C05498=1143.828,37.027,-50.516,-179.944,6.348,149.136
C05499=1143.823,37.277,-50.531,-179.940,6.350,149.135
C05500=1143.817,37.527,-50.546,-179.938,6.350,149.135
C05501=1143.813,37.776,-50.561,-179.936,6.352,149.135
C05502=1143.807,38.025,-50.576,-179.933,6.353,149.134
C05503=1143.802,38.275,-50.590,-179.930,6.354,149.133
C05504=1143.798,38.524,-50.605,-179.927,6.355,149.133
C05505=1143.792,38.774,-50.620,-179.925,6.355,149.132
C05506=1143.787,39.023,-50.635,-179.923,6.357,149.132
C05507=1143.782,39.272,-50.651,-179.920,6.358,149.131
C05508=1143.777,39.522,-50.665,-179.917,6.359,149.131
C05509=1143.772,39.771,-50.681,-179.915,6.360,149.130
C05510=1143.768,40.021,-50.696,-179.912,6.361,149.130
C05511=1143.762,40.271,-50.711,-179.910,6.362,149.129
C05512=1143.757,40.520,-50.726,-179.906,6.363,149.128
C05513=1143.752,40.770,-50.742,-179.904,6.364,149.128
C05514=1143.747,41.019,-50.757,-179.902,6.365,149.128
C05515=1143.742,41.269,-50.771,-179.899,6.366,149.127
C05516=1143.737,41.518,-50.786,-179.897,6.367,149.126
C05517=1143.732,41.767,-50.802,-179.894,6.369,149.126
C05518=1143.727,42.017,-50.816,-179.891,6.369,149.125
C05519=1143.722,42.267,-50.832,-179.888,6.371,149.125
C05520=1143.717,42.516,-50.847,-179.886,6.371,149.124
C05521=1143.712,42.766,-50.863,-179.883,6.373,149.124
C05522=1143.707,43.015,-50.878,-179.881,6.374,149.123
C05523=1143.701,43.265,-50.893,-179.878,6.375,149.123
C05524=1143.697,43.514,-50.908,-179.876,6.376,149.122
C05525=1143.691,43.763,-50.923,-179.873,6.378,149.122
C05526=1143.687,44.013,-50.939,-179.870,6.378,149.121
C05527=1143.682,44.263,-50.954,-179.868,6.379,149.121
C05528=1143.677,44.512,-50.970,-179.865,6.381,149.120
C05529=1143.672,44.762,-50.984,-179.863,6.381,149.120
C05530=1143.666,45.011,-51.000,-179.860,6.383,149.119
C05531=1143.662,45.260,-51.015,-179.857,6.383,149.118
C05532=1143.657,45.510,-51.031,-179.854,6.385,149.118
C05533=1143.651,45.760,-51.046,-179.852,6.386,149.117
C05534=1143.647,46.009,-51.061,-179.849,6.387,149.117
C05535=1143.641,46.258,-51.077,-179.847,6.388,149.116
C05536=1143.636,46.508,-51.092,-179.844,6.389,149.116
C05537=1143.632,46.757,-51.108,-179.841,6.390,149.115
C05538=1143.627,47.007,-51.123,-179.839,6.391,149.115
C05539=1143.621,47.256,-51.139,-179.837,6.392,149.114
C05540=1143.617,47.505,-51.154,-179.833,6.394,149.114
C05541=1143.611,47.755,-51.169,-179.831,6.394,149.113
C05542=1143.606,48.005,-51.185,-179.828,6.396,149.113
C05543=1143.602,48.254,-51.200,-179.826,6.396,149.112
C05544=1143.596,48.503,-51.216,-179.823,6.398,149.112
C05545=1143.591,48.753,-51.232,-179.820,6.399,149.111
C05546=1143.587,49.002,-51.247,-179.818,6.400,149.111
C05547=1143.582,49.252,-51.263,-179.815,6.401,149.110
C05548=1143.576,49.501,-51.278,-179.812,6.402,149.109
C05549=1143.571,49.750,-51.293,-179.810,6.403,149.109
C05550=1143.567,50.000,-51.309,-179.807,6.405,149.109
C05551=1143.561,50.250,-51.325,-179.805,6.405,149.108
C05552=1143.556,50.499,-51.340,-179.802,6.407,149.107
C05553=1143.551,50.748,-51.355,-179.800,6.408,149.107
C05554=1143.546,50.998,-51.371,-179.796,6.409,149.106
C05555=1143.541,51.248,-51.387,-179.794,6.410,149.106
C05556=1143.536,51.497,-51.402,-179.791,6.411,149.105
C05557=1143.532,51.747,-51.418,-179.789,6.412,149.105
C05558=1143.527,51.996,-51.434,-179.786,6.414,149.104
C05559=1143.521,52.245,-51.450,-179.783,6.415,149.104
C05560=1143.516,52.495,-51.466,-179.781,6.416,149.103
C05561=1143.511,52.745,-51.481,-179.778,6.417,149.103
C05562=1143.506,52.994,-51.496,-179.775,6.418,149.102
C05563=1143.501,53.262,-51.513,-179.773,6.420,149.102
C05564=1143.495,53.531,-51.530,-179.769,6.421,149.101
C05565=1143.490,53.800,-51.548,-179.767,6.422,149.101
C05566=1143.485,54.068,-51.565,-179.764,6.423,149.100
C05567=1143.479,54.318,-51.580,-179.761,6.425,149.099
C05568=1143.475,54.568,-51.596,-179.759,6.425,149.099
C05569=1143.469,54.817,-51.612,-179.756,6.427,149.098
C05570=1143.464,55.066,-51.628,-179.754,6.428,149.098
C05571=1143.460,55.316,-51.643,-179.751,6.429,149.098
C05572=1143.455,55.565,-51.659,-179.748,6.430,149.097
C05573=1143.450,55.814,-51.675,-179.746,6.431,149.096
C05574=1143.445,56.064,-51.691,-179.743,6.432,149.096
C05575=1143.439,56.314,-51.707,-179.740,6.433,149.095
C05576=1143.434,56.562,-51.723,-179.737,6.435,149.095
C05577=1143.430,56.812,-51.739,-179.735,6.436,149.094
C05578=1143.424,57.062,-51.755,-179.732,6.437,149.094
C05579=1143.420,57.311,-51.771,-179.730,6.438,149.093
C05580=1143.414,57.561,-51.787,-179.727,6.440,149.093
C05581=1143.409,57.810,-51.802,-179.724,6.440,149.092
C05582=1143.404,58.060,-51.819,-179.722,6.442,149.092
C05583=1143.400,58.309,-51.834,-179.719,6.443,149.091
C05584=1143.395,58.558,-51.851,-179.716,6.444,149.091
C05585=1143.390,58.808,-51.866,-179.714,6.446,149.090
C05586=1143.385,59.057,-51.882,-179.711,6.446,149.090
C05587=1143.380,59.307,-51.899,-179.708,6.448,149.089
C05588=1143.375,59.556,-51.914,-179.706,6.449,149.089
C05589=1143.370,59.805,-51.931,-179.703,6.450,149.088
C05590=1143.365,60.055,-51.946,-179.700,6.451,149.088
C05591=1143.360,60.304,-51.963,-179.698,6.452,149.087
C05592=1143.355,60.554,-51.979,-179.695,6.454,149.087
C05593=1143.350,60.803,-51.995,-179.693,6.454,149.086
C05594=1143.345,61.053,-52.011,-179.690,6.456,149.086
C05595=1143.339,61.302,-52.028,-179.687,6.458,149.085
C05596=1143.334,61.552,-52.044,-179.684,6.458,149.084
C05597=1143.329,61.801,-52.060,-179.682,6.460,149.084
C05598=1143.325,62.051,-52.076,-179.679,6.461,149.084
C05599=1143.319,62.299,-52.092,-179.676,6.462,149.083
C05600=1143.315,62.550,-52.108,-179.673,6.464,149.083
C05601=1143.310,62.798,-52.125,-179.671,6.465,149.082
C05602=1143.305,63.048,-52.141,-179.668,6.466,149.081
C05603=1143.300,63.297,-52.157,-179.666,6.467,149.081
C05604=1143.295,63.547,-52.174,-179.663,6.468,149.081
C05605=1143.290,63.796,-52.189,-179.660,6.470,149.080
C05606=1143.285,64.046,-52.206,-179.658,6.470,149.079
C05607=1143.280,64.295,-52.221,-179.655,6.472,149.079
C05608=1143.275,64.545,-52.239,-179.653,6.473,149.079
C05609=1143.270,64.794,-52.255,-179.650,6.474,149.078
C05610=1143.265,65.044,-52.271,-179.647,6.476,149.077
C05611=1143.260,65.293,-52.288,-179.645,6.477,149.077
C05612=1143.255,65.542,-52.304,-179.642,6.478,149.076
C05613=1143.251,65.792,-52.320,-179.639,6.480,149.076
C05614=1143.245,66.041,-52.337,-179.637,6.481,149.076
C05615=1143.240,66.291,-52.353,-179.633,6.482,149.075
C05616=1143.235,66.539,-52.370,-179.631,6.483,149.074
C05617=1143.230,66.790,-52.386,-179.629,6.484,149.074
C05618=1143.225,67.038,-52.402,-179.625,6.486,149.073
C05619=1143.221,67.288,-52.419,-179.623,6.486,149.073
C05620=1143.215,67.538,-52.435,-179.620,6.488,149.072
C05621=1143.210,67.787,-52.452,-179.618,6.490,149.072
C05622=1143.206,68.036,-52.468,-179.615,6.490,149.071
C05623=1143.201,68.285,-52.485,-179.612,6.492,149.071
C05624=1143.195,68.535,-52.502,-179.610,6.494,149.070
C05625=1143.191,68.785,-52.518,-179.607,6.494,149.070
C05626=1143.186,69.034,-52.534,-179.604,6.496,149.069
C05627=1143.181,69.283,-52.551,-179.601,6.497,149.069
C05628=1143.175,69.532,-52.568,-179.599,6.498,149.068
C05629=1143.171,69.782,-52.584,-179.596,6.499,149.068
C05630=1143.166,70.031,-52.601,-179.593,6.501,149.067
C05631=1143.161,70.281,-52.617,-179.591,6.502,149.067
C05632=1143.156,70.531,-52.634,-179.588,6.503,149.066
C05633=1143.151,70.780,-52.650,-179.586,6.504,149.066
C05634=1143.146,71.029,-52.667,-179.583,6.506,149.065
C05635=1143.141,71.279,-52.684,-179.580,6.507,149.065
C05636=1143.136,71.528,-52.701,-179.578,6.508,149.064
C05637=1143.131,71.777,-52.717,-179.575,6.510,149.064
C05638=1143.126,72.027,-52.734,-179.572,6.511,149.064
C05639=1143.122,72.276,-52.751,-179.569,6.513,149.063
C05640=1143.117,72.525,-52.767,-179.567,6.513,149.062
C05641=1143.111,72.775,-52.785,-179.564,6.515,149.062
C05642=1143.107,73.024,-52.801,-179.561,6.516,149.061
C05643=1143.102,73.273,-52.817,-179.559,6.517,149.061
C05644=1143.097,73.523,-52.835,-179.556,6.519,149.060
C05645=1143.092,73.772,-52.851,-179.553,6.521,149.060
C05646=1143.086,74.021,-52.868,-179.551,6.521,149.059
C05647=1143.082,74.271,-52.885,-179.548,6.523,149.059
C05648=1143.077,74.520,-52.902,-179.545,6.524,149.059
C05649=1143.072,74.770,-52.919,-179.543,6.525,149.058
C05650=1143.067,75.019,-52.935,-179.540,6.526,149.057
C05651=1143.062,75.269,-52.952,-179.537,6.528,149.057
C05652=1143.057,75.518,-52.969,-179.535,6.529,149.057
C05653=1143.052,75.767,-52.986,-179.532,6.530,149.056
C05654=1143.047,76.017,-53.003,-179.529,6.532,149.056
C05655=1143.043,76.266,-53.019,-179.526,6.534,149.055
C05656=1143.037,76.516,-53.037,-179.524,6.534,149.055
C05657=1143.032,76.765,-53.053,-179.521,6.536,149.054
C05658=1143.027,77.014,-53.071,-179.518,6.537,149.054
C05659=1143.023,77.264,-53.088,-179.516,6.538,149.053
C05660=1143.018,77.513,-53.105,-179.513,6.540,149.053
C05661=1143.013,77.762,-53.121,-179.510,6.541,149.052
C05662=1143.007,78.012,-53.138,-179.508,6.542,149.052
C05663=1143.003,78.261,-53.155,-179.505,6.544,149.051
C05664=1142.998,78.511,-53.173,-179.502,6.545,149.051
C05665=1142.993,78.759,-53.189,-179.499,6.547,149.050
C05666=1142.988,79.009,-53.207,-179.497,6.548,149.050
C05667=1142.982,79.278,-53.225,-179.494,6.549,149.049
C05668=1142.977,79.546,-53.243,-179.491,6.551,149.049
C05669=1142.972,79.815,-53.262,-179.488,6.552,149.048
C05670=1142.967,80.083,-53.281,-179.485,6.554,149.048
C05671=1142.962,80.333,-53.298,-179.482,6.555,149.047
C05672=1142.956,80.582,-53.315,-179.479,6.557,149.047
C05673=1142.952,80.831,-53.331,-179.477,6.558,149.046
C05674=1142.947,81.080,-53.349,-179.474,6.559,149.046
C05675=1142.942,81.330,-53.366,-179.471,6.561,149.045
C05676=1142.937,81.580,-53.383,-179.469,6.562,149.045
C05677=1142.932,81.829,-53.401,-179.466,6.563,149.044
C05678=1142.927,82.078,-53.418,-179.463,6.564,149.044
C05679=1142.922,82.327,-53.435,-179.460,6.566,149.043
C05680=1142.917,82.577,-53.453,-179.458,6.568,149.043
C05681=1142.913,82.826,-53.470,-179.456,6.569,149.042
C05682=1142.907,83.076,-53.487,-179.452,6.570,149.042
C05683=1142.903,83.325,-53.504,-179.450,6.572,149.041
C05684=1142.898,83.574,-53.521,-179.447,6.573,149.041
C05685=1142.892,83.823,-53.539,-179.445,6.574,149.040
C05686=1142.888,84.072,-53.556,-179.441,6.575,149.040
C05687=1142.883,84.322,-53.574,-179.439,6.577,149.039
C05688=1142.878,84.571,-53.591,-179.436,6.579,149.039
C05689=1142.873,84.821,-53.609,-179.434,6.580,149.039
C05690=1142.868,85.070,-53.626,-179.431,6.581,149.038
C05691=1142.863,85.320,-53.643,-179.428,6.583,149.037
C05692=1142.858,85.569,-53.661,-179.425,6.584,149.037
C05693=1142.854,85.819,-53.678,-179.423,6.585,149.037
C05694=1142.849,86.068,-53.696,-179.420,6.586,149.036
C05695=1142.844,86.317,-53.713,-179.417,6.588,149.036
C05696=1142.838,86.566,-53.730,-179.414,6.590,149.035
C05697=1142.834,86.815,-53.748,-179.412,6.591,149.035
C05698=1142.829,87.065,-53.765,-179.409,6.592,149.034
C05699=1142.824,87.314,-53.783,-179.406,6.594,149.034
C05700=1142.819,87.564,-53.800,-179.403,6.595,149.033
C05701=1142.814,87.813,-53.818,-179.401,6.597,149.033
C05702=1142.809,88.062,-53.835,-179.399,6.598,149.032
C05703=1142.804,88.311,-53.853,-179.395,6.599,149.032
C05704=1142.799,88.561,-53.871,-179.393,6.601,149.031
C05705=1142.794,88.810,-53.888,-179.390,6.603,149.031
C05706=1142.789,89.060,-53.906,-179.387,6.604,149.030
C05707=1142.785,89.308,-53.924,-179.385,6.605,149.030
C05708=1142.780,89.558,-53.941,-179.382,6.606,149.029
C05709=1142.775,89.807,-53.959,-179.379,6.608,149.029
C05710=1142.770,90.057,-53.977,-179.376,6.610,149.029
C05711=1142.765,90.306,-53.994,-179.374,6.611,149.028
C05712=1142.760,90.556,-54.012,-179.371,6.612,149.028
C05713=1142.755,90.805,-54.030,-179.368,6.614,149.027
C05714=1142.751,91.054,-54.047,-179.365,6.615,149.027
C05715=1142.746,91.303,-54.065,-179.363,6.617,149.026
C05716=1142.741,91.553,-54.083,-179.360,6.619,149.026
C05717=1142.736,91.802,-54.101,-179.357,6.620,149.025
C05718=1142.731,92.052,-54.118,-179.355,6.621,149.025
C05719=1142.726,92.301,-54.136,-179.352,6.622,149.024
C05720=1142.721,92.550,-54.154,-179.349,6.624,149.024
C05721=1142.716,92.799,-54.172,-179.346,6.626,149.023
C05722=1142.711,93.048,-54.190,-179.344,6.627,149.023
C05723=1142.706,93.298,-54.207,-179.341,6.628,149.022
C05724=1142.701,93.548,-54.225,-179.338,6.630,149.022
C05725=1142.697,93.797,-54.243,-179.336,6.631,149.022
C05726=1142.692,94.046,-54.261,-179.333,6.633,149.021
C05727=1142.687,94.295,-54.279,-179.330,6.635,149.021
C05728=1142.683,94.544,-54.297,-179.327,6.636,149.020
C05729=1142.678,94.793,-54.315,-179.324,6.638,149.020
C05730=1142.672,95.043,-54.332,-179.322,6.638,149.019
C05731=1142.668,95.292,-54.350,-179.319,6.640,149.019
C05732=1142.663,95.542,-54.368,-179.317,6.642,149.018
C05733=1142.657,95.791,-54.386,-179.313,6.643,149.018
C05734=1142.652,96.040,-54.404,-179.311,6.645,149.017
C05735=1142.648,96.290,-54.423,-179.308,6.646,149.017
C05736=1142.643,96.539,-54.441,-179.306,6.647,149.016
C05737=1142.638,96.789,-54.459,-179.303,6.649,149.016
C05738=1142.633,97.038,-54.477,-179.300,6.651,149.016
C05739=1142.628,97.287,-54.495,-179.297,6.652,149.015
C05740=1142.623,97.536,-54.513,-179.294,6.654,149.015
C05741=1142.618,97.785,-54.531,-179.292,6.655,149.014
C05742=1142.614,98.035,-54.549,-179.289,6.657,149.014
C05743=1142.609,98.284,-54.567,-179.287,6.658,149.013
C05744=1142.604,98.533,-54.585,-179.283,6.659,149.013
C05745=1142.599,98.783,-54.603,-179.281,6.661,149.012
C05746=1142.594,99.032,-54.621,-179.278,6.663,149.012
C05747=1142.589,99.281,-54.640,-179.275,6.664,149.011
C05748=1142.584,99.531,-54.658,-179.273,6.666,149.011
C05749=1142.579,99.780,-54.676,-179.270,6.668,149.011
C05750=1142.575,100.030,-54.694,-179.267,6.669,149.010
C05751=1142.570,100.278,-54.713,-179.264,6.670,149.010
C05752=1142.565,100.527,-54.730,-179.262,6.671,149.009
C05753=1142.560,100.776,-54.748,-179.259,6.673,149.009
C05754=1142.555,101.027,-54.767,-179.256,6.675,149.008
C05755=1142.550,101.276,-54.785,-179.253,6.677,149.008
C05756=1142.545,101.525,-54.803,-179.251,6.678,149.007
C05757=1142.540,101.774,-54.821,-179.248,6.680,149.007
C05758=1142.536,102.023,-54.840,-179.245,6.681,149.006
C05759=1142.531,102.273,-54.859,-179.242,6.683,149.006
C05760=1142.526,102.522,-54.877,-179.240,6.684,149.006
C05761=1142.521,102.771,-54.895,-179.237,6.685,149.005
C05762=1142.517,103.020,-54.914,-179.234,6.687,149.005
C05763=1142.512,103.270,-54.932,-179.231,6.688,149.004
C05764=1142.506,103.519,-54.951,-179.229,6.690,149.004
C05765=1142.501,103.768,-54.969,-179.226,6.692,149.003
C05766=1142.497,104.018,-54.988,-179.223,6.693,149.003
C05767=1142.492,104.267,-55.006,-179.220,6.695,149.002
C05768=1142.487,104.516,-55.024,-179.218,6.697,149.002
C05769=1142.482,104.765,-55.042,-179.215,6.699,149.002
C05770=1142.478,105.015,-55.061,-179.212,6.700,149.001
C05771=1142.472,105.283,-55.081,-179.209,6.702,149.001
C05772=1142.467,105.551,-55.101,-179.206,6.703,149.000
C05773=1142.461,105.819,-55.121,-179.203,6.705,149.000
C05774=1142.456,106.088,-55.141,-179.200,6.706,148.999
C05775=1142.451,106.338,-55.160,-179.198,6.708,148.999
C05776=1142.447,106.586,-55.178,-179.195,6.710,148.998
C05777=1142.442,106.836,-55.196,-179.192,6.711,148.998
C05778=1142.437,107.086,-55.215,-179.189,6.713,148.998
C05779=1142.432,107.334,-55.234,-179.187,6.715,148.997
C05780=1142.427,107.584,-55.252,-179.183,6.716,148.996
C05781=1142.422,107.833,-55.272,-179.181,6.718,148.996
C05782=1142.418,108.082,-55.290,-179.178,6.719,148.996
C05783=1142.413,108.331,-55.308,-179.175,6.721,148.995
C05784=1142.408,108.581,-55.327,-179.172,6.723,148.995
C05785=1142.403,108.830,-55.346,-179.170,6.724,148.994
C05786=1142.398,109.080,-55.365,-179.168,6.725,148.994
C05787=1142.394,109.328,-55.384,-179.165,6.727,148.994
C05788=1142.388,109.578,-55.402,-179.162,6.729,148.993
C05789=1142.384,109.827,-55.421,-179.159,6.730,148.993
C05790=1142.379,110.076,-55.439,-179.156,6.732,148.992
C05791=1142.374,110.325,-55.458,-179.153,6.733,148.992
C05792=1142.369,110.575,-55.477,-179.151,6.735,148.991
C05793=1142.364,110.824,-55.496,-179.148,6.737,148.991
C05794=1142.360,111.074,-55.514,-179.145,6.738,148.991
C05795=1142.354,111.323,-55.534,-179.143,6.740,148.990
C05796=1142.350,111.571,-55.552,-179.140,6.742,148.990
C05797=1142.345,111.821,-55.571,-179.137,6.743,148.989
C05798=1142.340,112.070,-55.590,-179.134,6.745,148.989
C05799=1142.335,112.319,-55.610,-179.131,6.746,148.988
C05800=1142.331,112.569,-55.628,-179.128,6.748,148.988
C05801=1142.326,112.818,-55.647,-179.126,6.750,148.987
C05802=1142.321,113.067,-55.665,-179.123,6.751,148.987
C05803=1142.316,113.316,-55.685,-179.120,6.753,148.987
C05804=1142.312,113.565,-55.704,-179.118,6.755,148.986
C05805=1142.306,113.814,-55.723,-179.115,6.757,148.986
C05806=1142.301,114.065,-55.742,-179.112,6.758,148.985
C05807=1142.297,114.313,-55.761,-179.109,6.760,148.985
C05808=1142.292,114.563,-55.780,-179.107,6.762,148.985
C05809=1142.287,114.812,-55.798,-179.103,6.763,148.984
C05810=1142.282,115.061,-55.818,-179.101,6.765,148.984
C05811=1142.277,115.310,-55.837,-179.098,6.766,148.983
C05812=1142.273,115.560,-55.856,-179.095,6.768,148.983
C05813=1142.267,115.808,-55.876,-179.093,6.770,148.982
C05814=1142.263,116.058,-55.894,-179.090,6.771,148.982
C05815=1142.258,116.307,-55.913,-179.087,6.773,148.982
C05816=1142.253,116.557,-55.933,-179.084,6.775,148.981
C05817=1142.248,116.805,-55.952,-179.082,6.776,148.981
C05818=1142.244,117.055,-55.971,-179.079,6.778,148.980
C05819=1142.238,117.304,-55.991,-179.076,6.780,148.980
C05820=1142.234,117.554,-56.009,-179.073,6.782,148.979
C05821=1142.229,117.802,-56.028,-179.071,6.783,148.979
C05822=1142.224,118.052,-56.048,-179.068,6.785,148.979
C05823=1142.219,118.301,-56.066,-179.065,6.786,148.978
C05824=1142.215,118.550,-56.086,-179.062,6.788,148.978
C05825=1142.209,118.799,-56.105,-179.059,6.790,148.977
C05826=1142.205,119.048,-56.125,-179.057,6.791,148.977
C05827=1142.201,119.298,-56.144,-179.054,6.793,148.976
C05828=1142.195,119.547,-56.163,-179.051,6.795,148.976
C05829=1142.190,119.796,-56.183,-179.048,6.796,148.976
C05830=1142.186,120.045,-56.202,-179.046,6.798,148.975
C05831=1142.181,120.294,-56.221,-179.043,6.800,148.975
C05832=1142.176,120.543,-56.241,-179.040,6.801,148.974
C05833=1142.171,120.793,-56.260,-179.038,6.803,148.974
C05834=1142.167,121.042,-56.279,-179.035,6.805,148.974
C05835=1142.162,121.291,-56.299,-179.032,6.807,148.973
C05836=1142.157,121.541,-56.318,-179.029,6.808,148.973
C05837=1142.152,121.790,-56.338,-179.027,6.810,148.972
C05838=1142.147,122.039,-56.357,-179.024,6.812,148.972
C05839=1142.143,122.288,-56.376,-179.021,6.813,148.972
C05840=1142.137,122.537,-56.396,-179.018,6.815,148.971
C05841=1142.133,122.787,-56.415,-179.015,6.818,148.971
C05842=1142.128,123.036,-56.435,-179.012,6.819,148.970
C05843=1142.123,123.284,-56.455,-179.010,6.821,148.970
C05844=1142.118,123.534,-56.475,-179.006,6.822,148.969
C05845=1142.114,123.783,-56.494,-179.004,6.824,148.969
C05846=1142.109,124.032,-56.513,-179.001,6.826,148.969
C05847=1142.104,124.282,-56.533,-178.998,6.827,148.968
C05848=1142.099,124.531,-56.552,-178.996,6.829,148.968
C05849=1142.094,124.780,-56.572,-178.993,6.831,148.967
C05850=1142.090,125.029,-56.592,-178.990,6.832,148.967
C05851=1142.085,125.279,-56.612,-178.987,6.834,148.967
C05852=1142.079,125.528,-56.631,-178.985,6.836,148.966
C05853=1142.075,125.777,-56.651,-178.982,6.837,148.966
C05854=1142.071,126.026,-56.670,-178.979,6.839,148.965
C05855=1142.066,126.275,-56.690,-178.976,6.842,148.965
C05856=1142.061,126.524,-56.709,-178.973,6.843,148.965
C05857=1142.057,126.773,-56.730,-178.970,6.845,148.964
C05858=1142.052,127.023,-56.749,-178.968,6.847,148.964
C05859=1142.046,127.272,-56.769,-178.965,6.848,148.963
C05860=1142.042,127.521,-56.788,-178.962,6.850,148.963
C05861=1142.037,127.770,-56.809,-178.960,6.852,148.963
C05862=1142.033,128.020,-56.828,-178.957,6.854,148.962
C05863=1142.027,128.269,-56.848,-178.954,6.855,148.962
C05864=1142.023,128.517,-56.868,-178.951,6.857,148.961
C05865=1142.018,128.767,-56.888,-178.949,6.859,148.961
C05866=1142.014,129.016,-56.908,-178.945,6.861,148.961
C05867=1142.008,129.265,-56.927,-178.943,6.863,148.960
C05868=1142.003,129.514,-56.947,-178.940,6.865,148.960
C05869=1141.999,129.763,-56.967,-178.937,6.866,148.959
C05870=1141.994,130.013,-56.987,-178.935,6.868,148.959
C05871=1141.989,130.261,-57.007,-178.932,6.870,148.959
C05872=1141.985,130.511,-57.027,-178.929,6.871,148.958
C05873=1141.979,130.760,-57.048,-178.926,6.873,148.958
C05874=1141.975,131.010,-57.067,-178.924,6.875,148.957
C05875=1141.970,131.278,-57.088,-178.920,6.877,148.957
C05876=1141.965,131.546,-57.110,-178.918,6.879,148.957
C05877=1141.959,131.815,-57.132,-178.914,6.881,148.956
C05878=1141.954,132.084,-57.153,-178.912,6.883,148.956
C05879=1141.949,132.332,-57.173,-178.909,6.885,148.956
C05880=1141.944,132.582,-57.193,-178.906,6.887,148.955
C05881=1141.940,132.831,-57.214,-178.903,6.888,148.955
C05882=1141.935,133.080,-57.234,-178.901,6.890,148.954
C05883=1141.930,133.329,-57.254,-178.897,6.892,148.954
C05884=1141.926,133.578,-57.274,-178.895,6.894,148.954
C05885=1141.921,133.828,-57.294,-178.892,6.896,148.953
C05886=1141.915,134.077,-57.314,-178.889,6.898,148.953
C05887=1141.911,134.326,-57.335,-178.887,6.899,148.952
C05888=1141.906,134.575,-57.354,-178.884,6.901,148.952
C05889=1141.902,134.824,-57.375,-178.881,6.903,148.952
C05890=1141.897,135.073,-57.395,-178.878,6.905,148.951
C05891=1141.892,135.323,-57.415,-178.875,6.907,148.951
C05892=1141.887,135.572,-57.436,-178.872,6.909,148.950
C05893=1141.883,135.821,-57.456,-178.870,6.910,148.950
C05894=1141.878,136.070,-57.475,-178.867,6.912,148.950
C05895=1141.873,136.319,-57.496,-178.864,6.914,148.949
C05896=1141.868,136.568,-57.517,-178.861,6.915,148.949
C05897=1141.864,136.817,-57.537,-178.859,6.918,148.949
C05898=1141.859,137.066,-57.557,-178.856,6.920,148.948
C05899=1141.854,137.316,-57.578,-178.853,6.922,148.948
C05900=1141.849,137.565,-57.598,-178.850,6.923,148.948
C05901=1141.845,137.814,-57.618,-178.848,6.925,148.947
C05902=1141.840,138.063,-57.638,-178.845,6.927,148.947
C05903=1141.835,138.312,-57.659,-178.842,6.929,148.946
C05904=1141.830,138.561,-57.679,-178.839,6.931,148.946
C05905=1141.826,138.810,-57.700,-178.836,6.933,148.946
C05906=1141.821,139.059,-57.721,-178.834,6.934,148.945
C05907=1141.816,139.308,-57.741,-178.831,6.936,148.945
C05908=1141.812,139.557,-57.761,-178.828,6.939,148.944
C05909=1141.806,139.807,-57.782,-178.825,6.940,148.944
C05910=1141.802,140.056,-57.802,-178.822,6.942,148.944
C05911=1141.797,140.304,-57.822,-178.819,6.944,148.943
C05912=1141.792,140.554,-57.843,-178.817,6.946,148.943
C05913=1141.787,140.803,-57.863,-178.814,6.948,148.943
C05914=1141.782,141.052,-57.884,-178.811,6.950,148.942
C05915=1141.778,141.301,-57.905,-178.808,6.952,148.942
C05916=1141.774,141.551,-57.925,-178.806,6.953,148.942
C05917=1141.769,141.800,-57.946,-178.803,6.955,148.941
C05918=1141.764,142.049,-57.967,-178.800,6.958,148.941
C05919=1141.759,142.298,-57.988,-178.797,6.959,148.940
C05920=1141.755,142.547,-58.008,-178.794,6.961,148.940
C05921=1141.750,142.796,-58.029,-178.792,6.963,148.940
C05922=1141.745,143.045,-58.050,-178.789,6.964,148.939
C05923=1141.741,143.294,-58.070,-178.786,6.967,148.939
C05924=1141.736,143.543,-58.091,-178.783,6.969,148.939
C05925=1141.731,143.792,-58.111,-178.781,6.971,148.938
C05926=1141.726,144.042,-58.132,-178.778,6.972,148.938
C05927=1141.721,144.291,-58.153,-178.775,6.974,148.938
C05928=1141.716,144.540,-58.174,-178.772,6.977,148.937
C05929=1141.712,144.788,-58.195,-178.769,6.978,148.937
C05930=1141.707,145.037,-58.216,-178.766,6.980,148.936
C05931=1141.703,145.286,-58.236,-178.764,6.982,148.936
C05932=1141.697,145.536,-58.257,-178.761,6.985,148.936
C05933=1141.694,145.785,-58.278,-178.758,6.986,148.935
C05934=1141.688,146.034,-58.299,-178.755,6.988,148.935
C05935=1141.683,146.284,-58.320,-178.753,6.990,148.935
C05936=1141.679,146.532,-58.341,-178.749,6.992,148.934
C05937=1141.674,146.781,-58.362,-178.747,6.994,148.934
C05938=1141.669,147.030,-58.382,-178.744,6.996,148.934
C05939=1141.664,147.280,-58.403,-178.741,6.997,148.933
C05940=1141.659,147.528,-58.425,-178.738,7.000,148.933
C05941=1141.655,147.777,-58.445,-178.736,7.002,148.933
C05942=1141.650,148.027,-58.466,-178.733,7.004,148.932
C05943=1141.646,148.276,-58.487,-178.730,7.005,148.932
C05944=1141.641,148.525,-58.508,-178.727,7.008,148.931
C05945=1141.636,148.774,-58.529,-178.724,7.010,148.931
C05946=1141.631,149.023,-58.550,-178.722,7.011,148.931
C05947=1141.627,149.272,-58.571,-178.719,7.014,148.931
C05948=1141.622,149.521,-58.593,-178.716,7.016,148.930
C05949=1141.618,149.770,-58.613,-178.713,7.018,148.930
C05950=1141.613,150.019,-58.635,-178.711,7.019,148.929
C05951=1141.608,150.268,-58.656,-178.708,7.021,148.929
C05952=1141.603,150.517,-58.676,-178.705,7.024,148.929
C05953=1141.598,150.766,-58.698,-178.702,7.025,148.928
C05954=1141.594,151.016,-58.719,-178.700,7.027,148.928
C05955=1141.589,151.265,-58.741,-178.697,7.029,148.928
C05956=1141.584,151.513,-58.761,-178.694,7.032,148.927
C05957=1141.579,151.763,-58.782,-178.691,7.033,148.927
C05958=1141.574,152.011,-58.804,-178.688,7.035,148.927
C05959=1141.570,152.261,-58.825,-178.685,7.038,148.926
C05960=1141.566,152.510,-58.846,-178.683,7.040,148.926
C05961=1141.560,152.759,-58.867,-178.680,7.041,148.926
C05962=1141.556,153.008,-58.889,-178.677,7.043,148.925
C05963=1141.551,153.258,-58.910,-178.674,7.046,148.925
C05964=1141.547,153.506,-58.931,-178.671,7.047,148.925
C05965=1141.542,153.755,-58.952,-178.669,7.049,148.924
C05966=1141.537,154.004,-58.974,-178.666,7.052,148.924
C05967=1141.533,154.253,-58.996,-178.663,7.054,148.924
C05968=1141.527,154.502,-59.017,-178.660,7.055,148.923
C05969=1141.523,154.751,-59.038,-178.657,7.058,148.923
C05970=1141.519,155.001,-59.059,-178.654,7.060,148.923
C05971=1141.514,155.249,-59.081,-178.652,7.062,148.922
C05972=1141.509,155.498,-59.103,-178.649,7.063,148.922
C05973=1141.504,155.747,-59.124,-178.646,7.066,148.922
C05974=1141.499,155.997,-59.146,-178.643,7.068,148.921
C05975=1141.494,156.246,-59.167,-178.641,7.069,148.921
C05976=1141.489,156.494,-59.188,-178.638,7.072,148.921
C05977=1141.486,156.743,-59.210,-178.635,7.074,148.920
C05978=1141.481,156.993,-59.231,-178.632,7.076,148.920
C05979=1141.476,157.261,-59.255,-178.629,7.078,148.920
C05980=1141.471,157.531,-59.278,-178.626,7.081,148.919
C05981=1141.465,157.800,-59.301,-178.623,7.082,148.919
C05982=1141.461,158.068,-59.325,-178.620,7.085,148.918
C05983=1141.456,158.317,-59.346,-178.617,7.087,148.918
C05984=1141.451,158.566,-59.367,-178.615,7.089,148.918
C05985=1141.447,158.816,-59.389,-178.612,7.091,148.918
C05986=1141.442,159.064,-59.411,-178.609,7.093,148.917
C05987=1141.437,159.314,-59.433,-178.606,7.095,148.917
C05988=1141.433,159.562,-59.455,-178.603,7.098,148.917
C05989=1141.427,159.811,-59.476,-178.601,7.099,148.916
C05990=1141.423,160.061,-59.498,-178.598,7.101,148.916
C05991=1141.418,160.309,-59.519,-178.595,7.104,148.916
C05992=1141.414,160.559,-59.541,-178.592,7.105,148.915
C05993=1141.409,160.807,-59.563,-178.589,7.108,148.915
C05994=1141.404,161.056,-59.585,-178.586,7.110,148.915
C05995=1141.400,161.305,-59.607,-178.584,7.112,148.914
C05996=1141.395,161.555,-59.628,-178.580,7.114,148.914
C05997=1141.391,161.804,-59.650,-178.578,7.116,148.914
C05998=1141.386,162.053,-59.672,-178.575,7.118,148.913
C05999=1141.380,162.302,-59.694,-178.572,7.120,148.913
C06000=1141.376,162.551,-59.716,-178.569,7.122,148.913
C06001=1141.371,162.800,-59.738,-178.567,7.124,148.913
C06002=1141.367,163.049,-59.760,-178.564,7.127,148.912
C06003=1141.362,163.298,-59.781,-178.561,7.128,148.912
C06004=1141.358,163.547,-59.803,-178.558,7.131,148.911
C06005=1141.353,163.796,-59.825,-178.556,7.133,148.911
C06006=1141.348,164.045,-59.847,-178.553,7.135,148.911
C06007=1141.344,164.293,-59.869,-178.550,7.137,148.911
C06008=1141.339,164.543,-59.891,-178.547,7.139,148.910
C06009=1141.334,164.792,-59.913,-178.545,7.141,148.910
C06010=1141.330,165.040,-59.936,-178.541,7.144,148.910
C06011=1141.325,165.289,-59.958,-178.539,7.145,148.909
C06012=1141.321,165.538,-59.980,-178.535,7.148,148.909
C06013=1141.316,165.787,-60.001,-178.533,7.150,148.909
C06014=1141.311,166.036,-60.023,-178.531,7.152,148.908
C06015=1141.306,166.285,-60.046,-178.527,7.154,148.908
C06016=1141.302,166.535,-60.068,-178.525,7.156,148.908
C06017=1141.297,166.783,-60.089,-178.522,7.159,148.908
C06018=1141.293,167.032,-60.112,-178.519,7.161,148.907
C06019=1141.287,167.281,-60.134,-178.516,7.162,148.907
C06020=1141.283,167.530,-60.156,-178.513,7.165,148.907
C06021=1141.278,167.779,-60.178,-178.511,7.167,148.906
C06022=1141.274,168.028,-60.200,-178.507,7.169,148.906
C06023=1141.269,168.277,-60.223,-178.505,7.172,148.906
C06024=1141.264,168.526,-60.245,-178.503,7.173,148.905
C06025=1141.260,168.775,-60.267,-178.499,7.176,148.905
C06026=1141.254,169.024,-60.290,-178.497,7.178,148.905
C06027=1141.250,169.273,-60.312,-178.494,7.180,148.905
C06028=1141.245,169.522,-60.334,-178.491,7.182,148.904
C06029=1141.241,169.771,-60.356,-178.488,7.185,148.904
C06030=1141.236,170.020,-60.379,-178.485,7.187,148.904
C06031=1141.232,170.269,-60.401,-178.483,7.188,148.903
C06032=1141.227,170.518,-60.423,-178.479,7.191,148.903
C06033=1141.222,170.766,-60.446,-178.477,7.193,148.903
C06034=1141.218,171.016,-60.468,-178.474,7.196,148.902
C06035=1141.213,171.265,-60.491,-178.471,7.197,148.902
C06036=1141.208,171.513,-60.513,-178.468,7.200,148.902
C06037=1141.204,171.763,-60.535,-178.466,7.202,148.902
C06038=1141.199,172.011,-60.558,-178.463,7.204,148.901
C06039=1141.194,172.260,-60.580,-178.460,7.207,148.901
C06040=1141.190,172.509,-60.604,-178.458,7.208,148.901
C06041=1141.185,172.758,-60.625,-178.454,7.211,148.900
C06042=1141.180,173.007,-60.647,-178.452,7.213,148.900
C06043=1141.176,173.256,-60.671,-178.449,7.215,148.900
C06044=1141.171,173.505,-60.692,-178.446,7.217,148.900
C06045=1141.166,173.754,-60.716,-178.443,7.220,148.899
C06046=1141.162,174.003,-60.738,-178.440,7.222,148.899
C06047=1141.157,174.252,-60.761,-178.437,7.224,148.899
C06048=1141.153,174.501,-60.784,-178.435,7.226,148.899
C06049=1141.148,174.750,-60.806,-178.432,7.228,148.898
C06050=1141.144,174.999,-60.829,-178.429,7.231,148.898
C06051=1141.138,175.248,-60.851,-178.427,7.233,148.898
C06052=1141.134,175.497,-60.874,-178.423,7.235,148.897
C06053=1141.129,175.746,-60.897,-178.421,7.237,148.897
C06054=1141.125,175.994,-60.919,-178.418,7.240,148.897
C06055=1141.120,176.243,-60.942,-178.415,7.242,148.896
C06056=1141.116,176.493,-60.964,-178.412,7.244,148.896
C06057=1141.111,176.742,-60.988,-178.410,7.246,148.896
C06058=1141.106,176.990,-61.010,-178.406,7.249,148.896
C06059=1141.101,177.239,-61.033,-178.404,7.251,148.895
C06060=1141.097,177.488,-61.056,-178.401,7.253,148.895
C06061=1141.093,177.737,-61.079,-178.398,7.255,148.895
C06062=1141.087,177.986,-61.101,-178.395,7.258,148.895
C06063=1141.083,178.235,-61.124,-178.393,7.260,148.894
C06064=1141.078,178.484,-61.147,-178.390,7.263,148.894
C06065=1141.074,178.733,-61.170,-178.387,7.264,148.894
C06066=1141.069,178.981,-61.192,-178.384,7.267,148.893
C06067=1141.064,179.230,-61.216,-178.382,7.269,148.893
C06068=1141.060,179.479,-61.239,-178.378,7.271,148.893
C06069=1141.055,179.728,-61.262,-178.376,7.274,148.893
C06070=1141.052,179.977,-61.285,-178.373,7.276,148.892
C06071=1141.046,180.226,-61.307,-178.370,7.278,148.892
C06072=1141.041,180.475,-61.330,-178.367,7.281,148.892
C06073=1141.037,180.724,-61.353,-178.365,7.282,148.892
C06074=1141.033,180.973,-61.376,-178.362,7.285,148.891
C06075=1141.028,181.222,-61.400,-178.359,7.287,148.891
C06076=1141.023,181.471,-61.423,-178.356,7.290,148.891
C06077=1141.019,181.719,-61.446,-178.354,7.292,148.891
C06078=1141.014,181.968,-61.469,-178.350,7.294,148.890
C06079=1141.009,182.217,-61.492,-178.348,7.296,148.890
C06080=1141.005,182.466,-61.514,-178.345,7.299,148.890
C06081=1141.000,182.715,-61.538,-178.342,7.301,148.889
C06082=1140.996,182.964,-61.561,-178.339,7.303,148.889
C06083=1140.991,183.233,-61.587,-178.336,7.306,148.889
C06084=1140.986,183.503,-61.611,-178.333,7.309,148.889
C06085=1140.981,183.773,-61.636,-178.331,7.311,148.888
C06086=1140.975,184.042,-61.661,-178.327,7.313,148.888
C06087=1140.971,184.291,-61.685,-178.324,7.316,148.888
C06088=1140.966,184.540,-61.708,-178.322,7.318,148.888
C06089=1140.962,184.789,-61.731,-178.318,7.320,148.887
C06090=1140.958,185.038,-61.755,-178.316,7.322,148.887
C06091=1140.953,185.287,-61.778,-178.313,7.325,148.887
C06092=1140.948,185.536,-61.802,-178.311,7.327,148.887
C06093=1140.943,185.785,-61.825,-178.307,7.330,148.886
C06094=1140.939,186.034,-61.848,-178.305,7.333,148.886
C06095=1140.935,186.282,-61.871,-178.302,7.334,148.886
C06096=1140.930,186.531,-61.894,-178.299,7.337,148.886
C06097=1140.925,186.781,-61.918,-178.296,7.339,148.885
C06098=1140.920,187.028,-61.941,-178.294,7.342,148.885
C06099=1140.916,187.277,-61.965,-178.291,7.344,148.885
C06100=1140.911,187.526,-61.988,-178.288,7.346,148.885
C06101=1140.906,187.775,-62.012,-178.285,7.348,148.884
C06102=1140.902,188.024,-62.035,-178.282,7.351,148.884
C06103=1140.897,188.273,-62.059,-178.279,7.354,148.884
C06104=1140.892,188.522,-62.082,-178.277,7.355,148.884
C06105=1140.888,188.771,-62.106,-178.274,7.358,148.883
C06106=1140.883,189.020,-62.129,-178.271,7.360,148.883
C06107=1140.879,189.268,-62.153,-178.268,7.363,148.883
C06108=1140.875,189.517,-62.176,-178.265,7.365,148.883
C06109=1140.870,189.766,-62.199,-178.263,7.367,148.883
C06110=1140.865,190.015,-62.223,-178.259,7.370,148.882
C06111=1140.861,190.263,-62.247,-178.257,7.372,148.882
C06112=1140.856,190.513,-62.270,-178.254,7.375,148.882
C06113=1140.851,190.761,-62.295,-178.252,7.377,148.882
C06114=1140.846,191.010,-62.318,-178.248,7.379,148.881
C06115=1140.842,191.259,-62.341,-178.246,7.382,148.881
C06116=1140.837,191.508,-62.365,-178.243,7.384,148.881
C06117=1140.833,191.757,-62.389,-178.240,7.387,148.881
C06118=1140.829,192.006,-62.413,-178.237,7.389,148.880
C06119=1140.824,192.255,-62.437,-178.235,7.391,148.880
C06120=1140.819,192.504,-62.460,-178.231,7.394,148.880
C06121=1140.815,192.752,-62.484,-178.229,7.396,148.880
C06122=1140.810,193.001,-62.507,-178.226,7.399,148.879
C06123=1140.806,193.250,-62.532,-178.224,7.401,148.879
C06124=1140.801,193.499,-62.555,-178.220,7.403,148.879
C06125=1140.797,193.747,-62.579,-178.218,7.406,148.879
C06126=1140.791,193.997,-62.603,-178.215,7.408,148.878
C06127=1140.787,194.245,-62.627,-178.212,7.411,148.878
C06128=1140.782,194.494,-62.650,-178.209,7.413,148.878
C06129=1140.779,194.743,-62.675,-178.207,7.415,148.878
C06130=1140.774,194.992,-62.699,-178.204,7.418,148.878
C06131=1140.769,195.241,-62.722,-178.201,7.420,148.877
C06132=1140.765,195.489,-62.746,-178.198,7.423,148.877
C06133=1140.760,195.738,-62.770,-178.195,7.426,148.877
C06134=1140.755,195.987,-62.794,-178.193,7.428,148.877
C06135=1140.751,196.235,-62.818,-178.189,7.430,148.876
C06136=1140.747,196.485,-62.842,-178.187,7.433,148.876
C06137=1140.742,196.733,-62.866,-178.184,7.435,148.876
C06138=1140.737,196.982,-62.891,-178.181,7.438,148.876
C06139=1140.732,197.231,-62.914,-178.178,7.441,148.876
C06140=1140.728,197.479,-62.938,-178.176,7.442,148.875
C06141=1140.724,197.728,-62.962,-178.173,7.445,148.875
C06142=1140.719,197.978,-62.987,-178.170,7.447,148.875
C06143=1140.714,198.226,-63.011,-178.167,7.450,148.875
C06144=1140.710,198.475,-63.035,-178.164,7.452,148.875
C06145=1140.706,198.723,-63.059,-178.162,7.454,148.874
C06146=1140.700,198.972,-63.083,-178.159,7.457,148.874
C06147=1140.696,199.222,-63.107,-178.156,7.460,148.874
C06148=1140.692,199.470,-63.131,-178.153,7.462,148.874
C06149=1140.687,199.719,-63.156,-178.150,7.465,148.873
C06150=1140.683,199.967,-63.180,-178.147,7.467,148.873
C06151=1140.678,200.217,-63.204,-178.145,7.469,148.873
C06152=1140.673,200.466,-63.229,-178.142,7.472,148.873
C06153=1140.669,200.714,-63.253,-178.139,7.475,148.873
C06154=1140.664,200.962,-63.277,-178.136,7.477,148.872
C06155=1140.660,201.212,-63.302,-178.134,7.480,148.872
C06156=1140.656,201.460,-63.326,-178.130,7.482,148.872
C06157=1140.651,201.709,-63.350,-178.128,7.484,148.872
C06158=1140.646,201.957,-63.375,-178.125,7.487,148.872
C06159=1140.642,202.207,-63.399,-178.122,7.490,148.871
C06160=1140.637,202.455,-63.424,-178.120,7.492,148.871
C06161=1140.633,202.704,-63.448,-178.117,7.494,148.871
C06162=1140.629,202.953,-63.472,-178.114,7.497,148.871
C06163=1140.624,203.202,-63.497,-178.111,7.500,148.871
C06164=1140.619,203.450,-63.521,-178.108,7.502,148.870
C06165=1140.614,203.699,-63.546,-178.105,7.505,148.870
C06166=1140.610,203.948,-63.570,-178.103,7.508,148.870
C06167=1140.605,204.196,-63.595,-178.100,7.509,148.870
C06168=1140.601,204.445,-63.619,-178.097,7.512,148.870
C06169=1140.596,204.694,-63.644,-178.094,7.515,148.869
C06170=1140.592,204.943,-63.668,-178.092,7.517,148.869
C06171=1140.587,205.191,-63.693,-178.089,7.520,148.869
C06172=1140.583,205.441,-63.717,-178.086,7.523,148.869
C06173=1140.578,205.689,-63.742,-178.083,7.525,148.869
C06174=1140.574,205.938,-63.766,-178.080,7.527,148.869
C06175=1140.569,206.187,-63.791,-178.077,7.530,148.868
C06176=1140.565,206.435,-63.816,-178.074,7.533,148.868
C06177=1140.560,206.684,-63.841,-178.072,7.535,148.868
C06178=1140.555,206.933,-63.865,-178.069,7.538,148.868
C06179=1140.551,207.181,-63.889,-178.066,7.541,148.868
C06180=1140.546,207.431,-63.914,-178.063,7.543,148.868
C06181=1140.542,207.679,-63.939,-178.061,7.545,148.867
C06182=1140.537,207.927,-63.964,-178.058,7.548,148.867
C06183=1140.533,208.177,-63.988,-178.055,7.551,148.867
C06184=1140.528,208.425,-64.013,-178.052,7.554,148.867
C06185=1140.524,208.674,-64.039,-178.050,7.556,148.867
C06186=1140.520,208.922,-64.063,-178.047,7.559,148.866
C06187=1140.514,209.194,-64.090,-178.043,7.561,148.866
C06188=1140.509,209.464,-64.117,-178.041,7.564,148.866
C06189=1140.505,209.735,-64.144,-178.037,7.567,148.866
C06190=1140.499,210.005,-64.171,-178.035,7.569,148.866
C06191=1140.495,210.254,-64.196,-178.032,7.572,148.865
C06192=1140.491,210.502,-64.221,-178.028,7.575,148.865
C06193=1140.486,210.752,-64.246,-178.026,7.578,148.865
C06194=1140.481,211.000,-64.271,-178.023,7.580,148.865
C06195=1140.477,211.249,-64.296,-178.020,7.582,148.865
C06196=1140.473,211.497,-64.320,-178.017,7.585,148.865
C06197=1140.468,211.746,-64.346,-178.015,7.588,148.864
C06198=1140.463,211.995,-64.371,-178.012,7.590,148.864
C06199=1140.460,212.243,-64.396,-178.009,7.593,148.864
C06200=1140.455,212.492,-64.421,-178.006,7.596,148.864
C06201=1140.450,212.741,-64.446,-178.003,7.599,148.864
C06202=1140.445,212.990,-64.471,-178.001,7.600,148.863
C06203=1140.441,213.239,-64.497,-177.998,7.603,148.863
C06204=1140.437,213.487,-64.521,-177.995,7.606,148.863
C06205=1140.432,213.736,-64.547,-177.992,7.609,148.863
C06206=1140.427,213.984,-64.571,-177.989,7.612,148.863
C06207=1140.423,214.233,-64.597,-177.987,7.614,148.863
C06208=1140.418,214.481,-64.622,-177.984,7.617,148.863
C06209=1140.414,214.730,-64.647,-177.981,7.620,148.862
C06210=1140.410,214.979,-64.673,-177.978,7.622,148.862
C06211=1140.405,215.228,-64.697,-177.976,7.624,148.862
C06212=1140.401,215.477,-64.723,-177.973,7.627,148.862
C06213=1140.396,215.725,-64.748,-177.970,7.630,148.862
C06214=1140.391,215.974,-64.773,-177.967,7.633,148.862
C06215=1140.387,216.222,-64.799,-177.964,7.636,148.861
C06216=1140.383,216.471,-64.824,-177.962,7.638,148.861
C06217=1140.379,216.720,-64.849,-177.959,7.641,148.861
C06218=1140.374,216.968,-64.874,-177.956,7.643,148.861
C06219=1140.370,217.217,-64.900,-177.953,7.646,148.861
C06220=1140.365,217.465,-64.925,-177.950,7.649,148.861
C06221=1140.360,217.715,-64.950,-177.948,7.651,148.861
C06222=1140.356,217.964,-64.976,-177.945,7.654,148.860
C06223=1140.351,218.212,-65.002,-177.942,7.657,148.860
C06224=1140.347,218.461,-65.027,-177.939,7.659,148.860
C06225=1140.342,218.710,-65.052,-177.936,7.662,148.860
C06226=1140.338,218.958,-65.078,-177.934,7.664,148.860
C06227=1140.333,219.207,-65.104,-177.931,7.667,148.860
C06228=1140.329,219.456,-65.129,-177.928,7.670,148.859
C06229=1140.324,219.704,-65.155,-177.925,7.673,148.859
C06230=1140.320,219.953,-65.180,-177.922,7.676,148.859
C06231=1140.316,220.201,-65.206,-177.920,7.679,148.859
C06232=1140.311,220.450,-65.231,-177.917,7.680,148.859
C06233=1140.307,220.699,-65.257,-177.914,7.683,148.859
C06234=1140.302,220.948,-65.282,-177.911,7.686,148.859
C06235=1140.297,221.196,-65.308,-177.908,7.689,148.859
C06236=1140.293,221.445,-65.333,-177.906,7.692,148.858
C06237=1140.289,221.693,-65.359,-177.902,7.695,148.858
C06238=1140.284,221.942,-65.385,-177.900,7.697,148.858
C06239=1140.280,222.190,-65.410,-177.897,7.700,148.858
C06240=1140.276,222.439,-65.436,-177.895,7.702,148.858
C06241=1140.270,222.688,-65.462,-177.892,7.705,148.858
C06242=1140.266,222.936,-65.488,-177.889,7.708,148.858
C06243=1140.262,223.185,-65.514,-177.886,7.711,148.857
C06244=1140.257,223.434,-65.539,-177.883,7.714,148.857
C06245=1140.253,223.682,-65.565,-177.881,7.716,148.857
C06246=1140.248,223.931,-65.590,-177.878,7.719,148.857
C06247=1140.245,224.179,-65.617,-177.875,7.722,148.857
C06248=1140.240,224.428,-65.643,-177.872,7.725,148.857
C06249=1140.235,224.676,-65.669,-177.869,7.727,148.857
C06250=1140.231,224.925,-65.694,-177.866,7.730,148.856
C06251=1140.226,225.174,-65.720,-177.863,7.733,148.856
C06252=1140.222,225.423,-65.746,-177.861,7.735,148.856
C06253=1140.217,225.672,-65.772,-177.858,7.738,148.856
C06254=1140.213,225.919,-65.798,-177.856,7.741,148.856
C06255=1140.208,226.168,-65.824,-177.852,7.743,148.856
C06256=1140.204,226.417,-65.850,-177.850,7.746,148.856
C06257=1140.200,226.666,-65.876,-177.847,7.749,148.856
C06258=1140.195,226.915,-65.902,-177.844,7.752,148.856
C06259=1140.190,227.162,-65.928,-177.842,7.754,148.855
C06260=1140.186,227.411,-65.954,-177.839,7.757,148.855
C06261=1140.181,227.660,-65.980,-177.836,7.760,148.855
C06262=1140.177,227.908,-66.007,-177.833,7.763,148.855
C06263=1140.173,228.157,-66.032,-177.830,7.766,148.855
C06264=1140.169,228.406,-66.058,-177.827,7.768,148.855
C06265=1140.163,228.654,-66.084,-177.824,7.771,148.855
C06266=1140.159,228.903,-66.111,-177.822,7.774,148.855
C06267=1140.155,229.151,-66.136,-177.819,7.777,148.854
C06268=1140.151,229.400,-66.163,-177.817,7.779,148.854
C06269=1140.146,229.649,-66.189,-177.814,7.782,148.854
C06270=1140.142,229.898,-66.215,-177.811,7.785,148.854
C06271=1140.137,230.146,-66.242,-177.808,7.788,148.854
C06272=1140.133,230.395,-66.268,-177.805,7.791,148.854
C06273=1140.128,230.643,-66.294,-177.802,7.794,148.854
C06274=1140.124,230.891,-66.320,-177.799,7.796,148.854
C06275=1140.120,231.140,-66.347,-177.797,7.799,148.854
C06276=1140.115,231.389,-66.373,-177.794,7.802,148.853
C06277=1140.111,231.637,-66.399,-177.791,7.805,148.853
C06278=1140.106,231.886,-66.426,-177.788,7.808,148.853
C06279=1140.102,232.134,-66.452,-177.786,7.810,148.853
C06280=1140.097,232.383,-66.479,-177.783,7.813,148.853
C06281=1140.093,232.632,-66.505,-177.780,7.816,148.853
C06282=1140.088,232.881,-66.531,-177.778,7.819,148.853
C06283=1140.084,233.129,-66.558,-177.774,7.821,148.853
C06284=1140.080,233.378,-66.584,-177.771,7.824,148.852
C06285=1140.075,233.626,-66.611,-177.769,7.827,148.852
C06286=1140.071,233.874,-66.637,-177.766,7.830,148.852
C06287=1140.066,234.123,-66.664,-177.763,7.833,148.852
C06288=1140.062,234.372,-66.691,-177.760,7.836,148.852
C06289=1140.058,234.620,-66.717,-177.757,7.839,148.852
C06290=1140.053,234.869,-66.743,-177.755,7.842,148.852
C06291=1140.049,235.141,-66.772,-177.752,7.845,148.852
C06292=1140.043,235.412,-66.801,-177.749,7.848,148.852
C06293=1140.038,235.684,-66.830,-177.746,7.851,148.852
C06294=1140.034,235.956,-66.859,-177.742,7.854,148.851
C06295=1140.030,236.205,-66.886,-177.740,7.857,148.851
C06296=1140.025,236.453,-66.913,-177.737,7.860,148.851
C06297=1140.021,236.702,-66.939,-177.734,7.863,148.851
C06298=1140.016,236.951,-66.966,-177.731,7.866,148.851
C06299=1140.011,237.199,-66.993,-177.728,7.869,148.851
C06300=1140.007,237.447,-67.020,-177.726,7.871,148.851
C06301=1140.003,237.696,-67.047,-177.723,7.874,148.851
C06302=1139.999,237.945,-67.073,-177.721,7.876,148.851
C06303=1139.994,238.193,-67.100,-177.718,7.879,148.851
C06304=1139.989,238.442,-67.127,-177.715,7.882,148.851
C06305=1139.985,238.690,-67.153,-177.712,7.885,148.851
C06306=1139.981,238.938,-67.180,-177.709,7.888,148.850
C06307=1139.976,239.187,-67.207,-177.707,7.891,148.850
C06308=1139.971,239.435,-67.234,-177.704,7.894,148.850
C06309=1139.968,239.684,-67.261,-177.701,7.897,148.850
C06310=1139.963,239.933,-67.288,-177.698,7.900,148.850
C06311=1139.958,240.182,-67.315,-177.695,7.903,148.850
C06312=1139.955,240.430,-67.341,-177.693,7.906,148.850
C06313=1139.950,240.678,-67.368,-177.690,7.909,148.850
C06314=1139.945,240.927,-67.395,-177.687,7.911,148.850
C06315=1139.941,241.175,-67.422,-177.684,7.914,148.850
C06316=1139.937,241.424,-67.449,-177.681,7.917,148.850
C06317=1139.933,241.672,-67.477,-177.679,7.920,148.850
C06318=1139.928,241.921,-67.504,-177.676,7.923,148.850
C06319=1139.924,242.169,-67.531,-177.673,7.926,148.849
C06320=1139.919,242.418,-67.558,-177.670,7.929,148.849
C06321=1139.915,242.666,-67.584,-177.667,7.932,148.849
C06322=1139.910,242.914,-67.612,-177.665,7.935,148.849
C06323=1139.906,243.163,-67.639,-177.662,7.938,148.849
C06324=1139.902,243.412,-67.666,-177.659,7.941,148.849
C06325=1139.897,243.661,-67.693,-177.656,7.944,148.849
C06326=1139.893,243.908,-67.721,-177.653,7.946,148.849
C06327=1139.889,244.157,-67.747,-177.651,7.949,148.849
C06328=1139.884,244.405,-67.774,-177.648,7.952,148.849
C06329=1139.880,244.654,-67.802,-177.645,7.955,148.849
C06330=1139.875,244.903,-67.829,-177.642,7.958,148.849
C06331=1139.871,245.151,-67.857,-177.639,7.961,148.849
C06332=1139.866,245.399,-67.884,-177.637,7.964,148.848
C06333=1139.862,245.648,-67.911,-177.634,7.967,148.848
C06334=1139.858,245.897,-67.938,-177.631,7.970,148.848
C06335=1139.853,246.145,-67.966,-177.628,7.973,148.848
C06336=1139.849,246.393,-67.993,-177.625,7.976,148.848
C06337=1139.844,246.642,-68.020,-177.623,7.979,148.848
C06338=1139.840,246.890,-68.048,-177.620,7.982,148.848
C06339=1139.836,247.139,-68.075,-177.618,7.985,148.848
C06340=1139.831,247.387,-68.102,-177.615,7.988,148.848
C06341=1139.827,247.636,-68.130,-177.612,7.991,148.848
C06342=1139.822,247.884,-68.158,-177.609,7.993,148.848
C06343=1139.818,248.133,-68.185,-177.606,7.996,148.848
C06344=1139.813,248.381,-68.212,-177.604,7.999,148.848
C06345=1139.809,248.630,-68.240,-177.601,8.002,148.848
C06346=1139.805,248.878,-68.268,-177.598,8.005,148.848
C06347=1139.800,249.126,-68.295,-177.595,8.008,148.848
C06348=1139.797,249.375,-68.323,-177.592,8.011,148.847
C06349=1139.792,249.623,-68.350,-177.590,8.014,148.847
C06350=1139.787,249.872,-68.377,-177.587,8.017,148.847
C06351=1139.784,250.120,-68.405,-177.584,8.020,148.847
C06352=1139.779,250.368,-68.433,-177.582,8.023,148.847
C06353=1139.775,250.617,-68.460,-177.579,8.026,148.847
C06354=1139.771,250.865,-68.488,-177.576,8.029,148.847
C06355=1139.766,251.114,-68.515,-177.573,8.032,148.847
C06356=1139.762,251.362,-68.543,-177.570,8.035,148.847
C06357=1139.757,251.611,-68.571,-177.567,8.038,148.847
C06358=1139.753,251.859,-68.599,-177.564,8.041,148.847
C06359=1139.748,252.107,-68.626,-177.561,8.044,148.847
C06360=1139.744,252.356,-68.654,-177.559,8.047,148.847
C06361=1139.740,252.604,-68.682,-177.556,8.050,148.847
C06362=1139.735,252.853,-68.709,-177.554,8.053,148.847
C06363=1139.731,253.101,-68.737,-177.551,8.056,148.847
C06364=1139.726,253.349,-68.765,-177.548,8.059,148.847
C06365=1139.722,253.599,-68.793,-177.545,8.062,148.847
C06366=1139.718,253.846,-68.820,-177.542,8.065,148.847
C06367=1139.714,254.094,-68.848,-177.540,8.068,148.847
C06368=1139.709,254.343,-68.877,-177.537,8.071,148.846
C06369=1139.705,254.592,-68.904,-177.534,8.074,148.847
C06370=1139.701,254.840,-68.932,-177.532,8.077,148.847
C06371=1139.696,255.088,-68.960,-177.529,8.080,148.846
C06372=1139.692,255.337,-68.989,-177.526,8.083,148.846
C06373=1139.688,255.585,-69.016,-177.523,8.087,148.846
C06374=1139.684,255.834,-69.044,-177.520,8.089,148.846
C06375=1139.678,256.082,-69.072,-177.517,8.092,148.846
C06376=1139.674,256.330,-69.100,-177.515,8.096,148.846
C06377=1139.670,256.579,-69.128,-177.512,8.099,148.846
C06378=1139.666,256.827,-69.156,-177.509,8.101,148.846
C06379=1139.661,257.075,-69.185,-177.506,8.104,148.846
C06380=1139.657,257.323,-69.212,-177.504,8.107,148.846
C06381=1139.653,257.572,-69.241,-177.501,8.110,148.846
C06382=1139.648,257.821,-69.268,-177.498,8.113,148.846
C06383=1139.644,258.069,-69.296,-177.496,8.116,148.846
C06384=1139.639,258.318,-69.325,-177.493,8.119,148.846
C06385=1139.635,258.566,-69.353,-177.489,8.123,148.846
C06386=1139.631,258.814,-69.381,-177.487,8.126,148.846
C06387=1139.627,259.063,-69.409,-177.484,8.129,148.846
C06388=1139.622,259.311,-69.437,-177.482,8.132,148.846
C06389=1139.618,259.560,-69.466,-177.479,8.135,148.846
C06390=1139.614,259.808,-69.494,-177.476,8.138,148.846
C06391=1139.610,260.056,-69.522,-177.473,8.141,148.846
C06392=1139.605,260.304,-69.551,-177.470,8.144,148.846
C06393=1139.601,260.552,-69.579,-177.468,8.147,148.846
C06394=1139.597,260.801,-69.608,-177.465,8.150,148.846
C06395=1139.592,261.074,-69.639,-177.462,8.154,148.846
C06396=1139.587,261.348,-69.670,-177.458,8.157,148.846
C06397=1139.582,261.622,-69.701,-177.456,8.160,148.846
C06398=1139.577,261.895,-69.733,-177.452,8.164,148.846
C06399=1139.574,262.144,-69.761,-177.450,8.167,148.846
C06400=1139.569,262.392,-69.789,-177.447,8.170,148.846
C06401=1139.565,262.640,-69.817,-177.444,8.173,148.846
C06402=1139.560,262.889,-69.846,-177.442,8.176,148.846
C06403=1139.556,263.137,-69.875,-177.439,8.179,148.846
C06404=1139.552,263.386,-69.903,-177.436,8.182,148.846
C06405=1139.547,263.634,-69.932,-177.434,8.185,148.846
C06406=1139.543,263.882,-69.960,-177.430,8.189,148.846
C06407=1139.538,264.130,-69.989,-177.427,8.192,148.846
C06408=1139.534,264.378,-70.017,-177.425,8.195,148.846
C06409=1139.530,264.627,-70.046,-177.422,8.198,148.846
C06410=1139.525,264.875,-70.075,-177.420,8.201,148.846
C06411=1139.521,265.123,-70.103,-177.417,8.204,148.846
C06412=1139.517,265.372,-70.132,-177.414,8.207,148.846
C06413=1139.513,265.620,-70.160,-177.412,8.210,148.846
C06414=1139.508,265.868,-70.189,-177.408,8.214,148.846
C06415=1139.504,266.117,-70.218,-177.405,8.217,148.846
C06416=1139.500,266.365,-70.246,-177.403,8.220,148.846
C06417=1139.495,266.614,-70.275,-177.400,8.223,148.846
C06418=1139.491,266.862,-70.305,-177.398,8.226,148.846
C06419=1139.486,267.110,-70.333,-177.395,8.229,148.846
C06420=1139.483,267.358,-70.362,-177.392,8.233,148.846
C06421=1139.478,267.607,-70.391,-177.389,8.236,148.846
C06422=1139.474,267.855,-70.420,-177.386,8.239,148.846
C06423=1139.470,268.103,-70.448,-177.383,8.242,148.846
C06424=1139.465,268.351,-70.477,-177.381,8.245,148.846
C06425=1139.461,268.600,-70.506,-177.378,8.248,148.846
C06426=1139.457,268.848,-70.535,-177.376,8.251,148.846
C06427=1139.452,269.096,-70.563,-177.373,8.255,148.846
C06428=1139.448,269.345,-70.593,-177.370,8.258,148.846
C06429=1139.444,269.593,-70.621,-177.367,8.261,148.846
C06430=1139.440,269.842,-70.651,-177.364,8.264,148.846
C06431=1139.435,270.089,-70.680,-177.362,8.267,148.846
C06432=1139.431,270.338,-70.708,-177.359,8.270,148.846
C06433=1139.427,270.586,-70.738,-177.356,8.273,148.846
C06434=1139.423,270.834,-70.767,-177.353,8.277,148.846
C06435=1139.418,271.083,-70.795,-177.351,8.280,148.846
C06436=1139.413,271.331,-70.825,-177.348,8.283,148.846
C06437=1139.409,271.579,-70.854,-177.345,8.286,148.846
C06438=1139.405,271.828,-70.882,-177.342,8.290,148.846
C06439=1139.401,272.076,-70.912,-177.339,8.292,148.846
C06440=1139.397,272.324,-70.941,-177.337,8.296,148.846
C06441=1139.392,272.572,-70.970,-177.334,8.299,148.846
C06442=1139.388,272.821,-70.999,-177.331,8.302,148.846
C06443=1139.384,273.069,-71.029,-177.329,8.305,148.846
C06444=1139.379,273.317,-71.058,-177.326,8.309,148.846
C06445=1139.375,273.565,-71.087,-177.323,8.311,148.846
C06446=1139.371,273.814,-71.117,-177.321,8.315,148.846
C06447=1139.366,274.062,-71.145,-177.318,8.318,148.846
C06448=1139.362,274.310,-71.175,-177.315,8.321,148.846
C06449=1139.358,274.558,-71.204,-177.312,8.325,148.846
C06450=1139.354,274.806,-71.233,-177.309,8.328,148.846
C06451=1139.350,275.055,-71.263,-177.306,8.331,148.846
C06452=1139.346,275.303,-71.292,-177.304,8.334,148.846
C06453=1139.342,275.551,-71.321,-177.301,8.337,148.846
C06454=1139.337,275.799,-71.351,-177.298,8.340,148.846
C06455=1139.333,276.048,-71.380,-177.296,8.344,148.846
C06456=1139.329,276.295,-71.409,-177.293,8.347,148.846
C06457=1139.324,276.544,-71.439,-177.290,8.350,148.846
C06458=1139.320,276.792,-71.468,-177.288,8.353,148.846
C06459=1139.315,277.040,-71.498,-177.284,8.357,148.846
C06460=1139.311,277.289,-71.528,-177.282,8.360,148.847
C06461=1139.307,277.537,-71.557,-177.279,8.363,148.846
C06462=1139.303,277.785,-71.587,-177.277,8.366,148.847
C06463=1139.299,278.033,-71.616,-177.273,8.370,148.847
C06464=1139.294,278.282,-71.646,-177.271,8.373,148.847
C06465=1139.290,278.530,-71.675,-177.268,8.376,148.847
C06466=1139.286,278.778,-71.705,-177.266,8.379,148.847
C06467=1139.282,279.027,-71.734,-177.263,8.382,148.847
C06468=1139.278,279.274,-71.764,-177.260,8.386,148.847
C06469=1139.274,279.522,-71.794,-177.257,8.389,148.847
C06470=1139.269,279.771,-71.824,-177.255,8.392,148.847
C06471=1139.265,280.019,-71.853,-177.252,8.395,148.847
C06472=1139.260,280.268,-71.883,-177.249,8.399,148.847
C06473=1139.256,280.516,-71.912,-177.246,8.402,148.847
C06474=1139.252,280.763,-71.942,-177.244,8.405,148.847
C06475=1139.247,281.012,-71.972,-177.241,8.408,148.847
C06476=1139.243,281.260,-72.002,-177.238,8.412,148.847
C06477=1139.239,281.509,-72.031,-177.235,8.415,148.847
C06478=1139.235,281.756,-72.061,-177.233,8.418,148.847
C06479=1139.231,282.005,-72.091,-177.230,8.421,148.847
C06480=1139.226,282.253,-72.121,-177.227,8.425,148.847
C06481=1139.222,282.501,-72.151,-177.225,8.428,148.848
C06482=1139.218,282.749,-72.180,-177.222,8.431,148.847
C06483=1139.213,282.998,-72.210,-177.219,8.434,148.848
C06484=1139.209,283.245,-72.241,-177.216,8.438,148.848
C06485=1139.205,283.493,-72.270,-177.214,8.441,148.848
C06486=1139.201,283.742,-72.300,-177.211,8.444,148.848
C06487=1139.196,283.990,-72.330,-177.209,8.448,148.848
C06488=1139.192,284.238,-72.360,-177.205,8.451,148.848
C06489=1139.188,284.486,-72.390,-177.202,8.454,148.848
C06490=1139.184,284.735,-72.420,-177.200,8.458,148.848
C06491=1139.180,284.983,-72.451,-177.197,8.460,148.848
C06492=1139.176,285.231,-72.480,-177.194,8.465,148.848
C06493=1139.171,285.479,-72.511,-177.192,8.467,148.848
C06494=1139.167,285.727,-72.540,-177.189,8.471,148.848
C06495=1139.162,285.975,-72.571,-177.186,8.474,148.848
C06496=1139.158,286.223,-72.600,-177.183,8.478,148.848
C06497=1139.154,286.471,-72.631,-177.181,8.481,148.848
C06498=1139.150,286.720,-72.661,-177.178,8.484,148.849
C06499=1139.145,286.995,-72.694,-177.175,8.488,148.849
C06500=1139.141,287.271,-72.729,-177.172,8.492,148.849
C06501=1139.136,287.546,-72.761,-177.169,8.495,148.849
C06502=1139.132,287.822,-72.795,-177.166,8.499,148.849
C06503=1139.127,288.070,-72.826,-177.163,8.502,148.849
C06504=1139.123,288.318,-72.855,-177.161,8.506,148.849
C06505=1139.119,288.567,-72.886,-177.158,8.509,148.849
C06506=1139.115,288.814,-72.916,-177.155,8.513,148.849
C06507=1139.110,289.063,-72.946,-177.153,8.516,148.849
C06508=1139.106,289.310,-72.977,-177.150,8.519,148.849
C06509=1139.102,289.558,-73.007,-177.147,8.523,148.850
C06510=1139.098,289.807,-73.037,-177.144,8.526,148.850
C06511=1139.093,290.055,-73.068,-177.142,8.529,148.850
C06512=1139.090,290.303,-73.098,-177.139,8.532,148.850
C06513=1139.085,290.551,-73.129,-177.136,8.536,148.850
C06514=1139.081,290.799,-73.159,-177.133,8.539,148.850
C06515=1139.077,291.048,-73.189,-177.131,8.542,148.850
C06516=1139.072,291.296,-73.220,-177.128,8.546,148.850
C06517=1139.068,291.543,-73.250,-177.125,8.549,148.850
C06518=1139.064,291.791,-73.281,-177.123,8.553,148.850
C06519=1139.060,292.040,-73.312,-177.119,8.556,148.850
C06520=1139.056,292.288,-73.342,-177.117,8.560,148.850
C06521=1139.051,292.536,-73.373,-177.115,8.563,148.851
C06522=1139.048,292.784,-73.404,-177.111,8.567,148.851
C06523=1139.043,293.033,-73.434,-177.109,8.570,148.851
C06524=1139.039,293.280,-73.464,-177.106,8.573,148.851
C06525=1139.034,293.528,-73.495,-177.103,8.577,148.851
C06526=1139.030,293.777,-73.526,-177.101,8.580,148.851
C06527=1139.027,294.024,-73.556,-177.098,8.583,148.851
C06528=1139.022,294.272,-73.587,-177.095,8.587,148.851
C06529=1139.018,294.521,-73.618,-177.093,8.590,148.851
C06530=1139.014,294.769,-73.648,-177.090,8.593,148.851
C06531=1139.009,295.017,-73.679,-177.087,8.597,148.852
C06532=1139.005,295.265,-73.710,-177.084,8.600,148.852
C06533=1139.001,295.513,-73.741,-177.082,8.604,148.852
C06534=1138.997,295.760,-73.772,-177.079,8.608,148.852
C06535=1138.993,296.009,-73.803,-177.076,8.611,148.852
C06536=1138.989,296.257,-73.834,-177.074,8.614,148.852
C06537=1138.985,296.506,-73.865,-177.071,8.618,148.852
C06538=1138.981,296.753,-73.895,-177.068,8.621,148.852
C06539=1138.976,297.001,-73.926,-177.066,8.624,148.852
C06540=1138.972,297.249,-73.957,-177.063,8.628,148.853
C06541=1138.968,297.497,-73.988,-177.060,8.631,148.853
C06542=1138.963,297.745,-74.019,-177.058,8.634,148.853
C06543=1138.960,297.994,-74.050,-177.055,8.638,148.853
C06544=1138.955,298.241,-74.080,-177.052,8.641,148.853
C06545=1138.952,298.490,-74.112,-177.050,8.645,148.853
C06546=1138.947,298.737,-74.143,-177.047,8.649,148.853
C06547=1138.942,298.985,-74.174,-177.044,8.652,148.853
C06548=1138.938,299.234,-74.205,-177.041,8.656,148.854
C06549=1138.935,299.481,-74.236,-177.039,8.659,148.854
C06550=1138.931,299.730,-74.267,-177.036,8.662,148.854
C06551=1138.926,299.978,-74.298,-177.033,8.666,148.854
C06552=1138.922,300.226,-74.329,-177.031,8.669,148.854
C06553=1138.918,300.474,-74.360,-177.029,8.672,148.854
C06554=1138.913,300.722,-74.391,-177.025,8.676,148.854
C06555=1138.910,300.970,-74.423,-177.023,8.679,148.854
C06556=1138.905,301.218,-74.454,-177.020,8.684,148.855
C06557=1138.901,301.466,-74.485,-177.017,8.686,148.855
C06558=1138.897,301.714,-74.516,-177.015,8.690,148.855
C06559=1138.893,301.962,-74.548,-177.012,8.694,148.855
C06560=1138.888,302.210,-74.579,-177.009,8.697,148.855
C06561=1138.885,302.458,-74.611,-177.007,8.700,148.855
C06562=1138.880,302.706,-74.641,-177.004,8.704,148.855
C06563=1138.876,302.954,-74.673,-177.001,8.707,148.856
C06564=1138.872,303.202,-74.704,-176.999,8.711,148.856
C06565=1138.868,303.450,-74.736,-176.996,8.714,148.856
C06566=1138.863,303.698,-74.767,-176.993,8.718,148.856
C06567=1138.860,303.946,-74.798,-176.990,8.722,148.856
C06568=1138.855,304.194,-74.829,-176.988,8.725,148.856
C06569=1138.851,304.442,-74.861,-176.985,8.729,148.856
C06570=1138.847,304.690,-74.892,-176.982,8.732,148.856
C06571=1138.843,304.938,-74.924,-176.980,8.735,148.857
C06572=1138.839,305.185,-74.955,-176.977,8.739,148.857
C06573=1138.835,305.434,-74.986,-176.975,8.742,148.857
C06574=1138.830,305.682,-75.019,-176.971,8.746,148.857
C06575=1138.826,305.929,-75.050,-176.969,8.749,148.857
C06576=1138.822,306.178,-75.081,-176.967,8.753,148.857
C06577=1138.818,306.425,-75.113,-176.964,8.757,148.858
C06578=1138.814,306.673,-75.145,-176.961,8.760,148.858
C06579=1138.810,306.921,-75.176,-176.959,8.764,148.858
C06580=1138.806,307.169,-75.207,-176.956,8.767,148.858
C06581=1138.801,307.418,-75.240,-176.953,8.771,148.858
C06582=1138.797,307.665,-75.271,-176.950,8.774,148.858
C06583=1138.793,307.913,-75.303,-176.948,8.778,148.859
C06584=1138.789,308.162,-75.334,-176.945,8.782,148.859
C06585=1138.785,308.409,-75.366,-176.942,8.785,148.859
C06586=1138.780,308.657,-75.398,-176.939,8.789,148.859
C06587=1138.776,308.905,-75.430,-176.937,8.792,148.859
C06588=1138.772,309.153,-75.461,-176.934,8.796,148.859
C06589=1138.769,309.401,-75.493,-176.932,8.799,148.860
C06590=1138.764,309.649,-75.525,-176.930,8.803,148.860
C06591=1138.760,309.897,-75.557,-176.927,8.807,148.860
C06592=1138.756,310.145,-75.589,-176.924,8.810,148.860
C06593=1138.752,310.393,-75.620,-176.921,8.814,148.860
C06594=1138.747,310.641,-75.652,-176.919,8.817,148.860
C06595=1138.743,310.889,-75.684,-176.916,8.821,148.861
C06596=1138.739,311.136,-75.716,-176.913,8.824,148.861
C06597=1138.735,311.385,-75.748,-176.910,8.828,148.861
C06598=1138.731,311.633,-75.780,-176.908,8.832,148.861
C06599=1138.727,311.880,-75.811,-176.905,8.836,148.861
C06600=1138.722,312.128,-75.844,-176.903,8.839,148.861
C06601=1138.719,312.376,-75.876,-176.900,8.842,148.862
C06602=1138.715,312.624,-75.908,-176.897,8.846,148.862
C06603=1138.710,312.902,-75.944,-176.894,8.850,148.862
C06604=1138.705,313.180,-75.979,-176.891,8.854,148.862
C06605=1138.700,313.458,-76.015,-176.888,8.858,148.862
C06606=1138.696,313.736,-76.052,-176.885,8.862,148.863
C06607=1138.692,313.984,-76.083,-176.883,8.865,148.863
C06608=1138.688,314.232,-76.115,-176.880,8.869,148.863
C06609=1138.684,314.479,-76.148,-176.878,8.873,148.863
C06610=1138.680,314.727,-76.180,-176.875,8.877,148.863
C06611=1138.676,314.976,-76.213,-176.872,8.880,148.864
C06612=1138.671,315.223,-76.244,-176.869,8.884,148.864
C06613=1138.667,315.471,-76.277,-176.867,8.887,148.864
C06614=1138.663,315.719,-76.309,-176.864,8.891,148.864
C06615=1138.659,315.967,-76.342,-176.862,8.895,148.864
C06616=1138.655,316.215,-76.373,-176.859,8.899,148.865
C06617=1138.651,316.462,-76.406,-176.857,8.902,148.865
C06618=1138.647,316.710,-76.438,-176.854,8.906,148.865
C06619=1138.642,316.959,-76.471,-176.851,8.909,148.865
C06620=1138.639,317.206,-76.503,-176.848,8.913,148.865
C06621=1138.635,317.454,-76.536,-176.846,8.917,148.866
C06622=1138.630,317.702,-76.567,-176.843,8.921,148.866
C06623=1138.626,317.949,-76.600,-176.841,8.924,148.866
C06624=1138.622,318.198,-76.632,-176.838,8.928,148.866
C06625=1138.618,318.445,-76.665,-176.836,8.931,148.866
C06626=1138.615,318.693,-76.697,-176.833,8.935,148.867
C06627=1138.610,318.941,-76.730,-176.830,8.939,148.867
C06628=1138.606,319.189,-76.763,-176.827,8.943,148.867
C06629=1138.603,319.437,-76.795,-176.825,8.946,148.867
C06630=1138.598,319.684,-76.827,-176.822,8.950,148.867
C06631=1138.594,319.932,-76.860,-176.820,8.953,148.868
C06632=1138.590,320.180,-76.892,-176.817,8.957,148.868
C06633=1138.586,320.428,-76.925,-176.814,8.961,148.868
C06634=1138.582,320.676,-76.957,-176.811,8.965,148.868
C06635=1138.578,320.924,-76.990,-176.809,8.968,148.868
C06636=1138.573,321.172,-77.023,-176.806,8.972,148.869
C06637=1138.570,321.419,-77.055,-176.804,8.975,148.869
C06638=1138.566,321.667,-77.089,-176.801,8.979,148.869
C06639=1138.561,321.916,-77.121,-176.799,8.983,148.869
C06640=1138.558,322.163,-77.154,-176.796,8.987,148.870
C06641=1138.553,322.411,-77.186,-176.793,8.990,148.870
C06642=1138.549,322.659,-77.219,-176.790,8.994,148.870
C06643=1138.546,322.906,-77.252,-176.788,8.997,148.870
C06644=1138.542,323.154,-77.285,-176.786,9.002,148.871
C06645=1138.537,323.403,-77.317,-176.783,9.006,148.871
C06646=1138.533,323.650,-77.351,-176.780,9.009,148.871
C06647=1138.530,323.898,-77.383,-176.777,9.013,148.871
C06648=1138.526,324.145,-77.416,-176.775,9.016,148.871
C06649=1138.521,324.394,-77.449,-176.772,9.020,148.872
C06650=1138.517,324.641,-77.482,-176.770,9.024,148.872
C06651=1138.513,324.889,-77.515,-176.767,9.028,148.872
C06652=1138.509,325.137,-77.548,-176.764,9.031,148.872
C06653=1138.505,325.384,-77.581,-176.762,9.035,148.873
C06654=1138.501,325.633,-77.613,-176.760,9.039,148.873
C06655=1138.497,325.880,-77.646,-176.757,9.043,148.873
C06656=1138.493,326.128,-77.680,-176.754,9.047,148.873
C06657=1138.488,326.376,-77.713,-176.751,9.050,148.874
C06658=1138.484,326.624,-77.746,-176.748,9.054,148.874
C06659=1138.481,326.871,-77.778,-176.746,9.057,148.874
C06660=1138.477,327.119,-77.812,-176.744,9.062,148.874
C06661=1138.473,327.367,-77.845,-176.741,9.065,148.875
C06662=1138.469,327.614,-77.878,-176.738,9.069,148.875
C06663=1138.464,327.862,-77.911,-176.735,9.073,148.875
C06664=1138.460,328.110,-77.944,-176.733,9.076,148.875
C06665=1138.456,328.357,-77.977,-176.730,9.080,148.875
C06666=1138.452,328.605,-78.010,-176.728,9.084,148.876
C06667=1138.448,328.853,-78.044,-176.725,9.088,148.876
C06668=1138.444,329.101,-78.077,-176.723,9.091,148.876
C06669=1138.440,329.348,-78.110,-176.720,9.095,148.877
C06670=1138.436,329.597,-78.143,-176.717,9.100,148.877
C06671=1138.432,329.845,-78.177,-176.715,9.103,148.877
C06672=1138.428,330.092,-78.210,-176.712,9.107,148.877
C06673=1138.424,330.340,-78.243,-176.710,9.110,148.878
C06674=1138.420,330.587,-78.277,-176.707,9.114,148.878
C06675=1138.416,330.835,-78.310,-176.704,9.119,148.878
C06676=1138.412,331.083,-78.343,-176.702,9.122,148.878
C06677=1138.408,331.331,-78.377,-176.699,9.126,148.879
C06678=1138.404,331.579,-78.410,-176.697,9.129,148.879
C06679=1138.400,331.826,-78.443,-176.694,9.134,148.879
C06680=1138.396,332.074,-78.477,-176.691,9.138,148.880
C06681=1138.392,332.321,-78.510,-176.689,9.141,148.880
C06682=1138.387,332.569,-78.544,-176.686,9.145,148.880
C06683=1138.383,332.818,-78.577,-176.684,9.149,148.880
C06684=1138.379,333.065,-78.611,-176.681,9.153,148.881
C06685=1138.375,333.313,-78.644,-176.678,9.157,148.881
C06686=1138.371,333.560,-78.677,-176.676,9.160,148.881
C06687=1138.367,333.807,-78.711,-176.673,9.165,148.881
C06688=1138.364,334.056,-78.745,-176.671,9.168,148.882
C06689=1138.360,334.304,-78.778,-176.668,9.172,148.882
C06690=1138.355,334.551,-78.812,-176.666,9.176,148.882
C06691=1138.351,334.799,-78.846,-176.663,9.180,148.883
C06692=1138.347,335.046,-78.879,-176.660,9.184,148.883
C06693=1138.344,335.294,-78.913,-176.658,9.187,148.883
C06694=1138.340,335.541,-78.947,-176.656,9.191,148.883
C06695=1138.335,335.789,-78.981,-176.653,9.195,148.884
C06696=1138.331,336.037,-79.014,-176.650,9.199,148.884
C06697=1138.328,336.285,-79.048,-176.648,9.203,148.884
C06698=1138.324,336.532,-79.082,-176.645,9.207,148.885
C06699=1138.319,336.780,-79.116,-176.643,9.210,148.885
C06700=1138.316,337.028,-79.150,-176.640,9.215,148.885
C06701=1138.311,337.276,-79.183,-176.637,9.219,148.885
C06702=1138.308,337.523,-79.217,-176.635,9.222,148.886
C06703=1138.303,337.771,-79.251,-176.632,9.226,148.886
C06704=1138.300,338.019,-79.285,-176.630,9.230,148.886
C06705=1138.295,338.266,-79.318,-176.627,9.234,148.887
C06706=1138.291,338.514,-79.352,-176.624,9.238,148.887
C06707=1138.287,338.795,-79.391,-176.622,9.242,148.887
C06708=1138.283,339.075,-79.429,-176.619,9.247,148.888
C06709=1138.278,339.356,-79.468,-176.615,9.251,148.888
C06710=1138.273,339.637,-79.506,-176.613,9.256,148.888
C06711=1138.269,339.884,-79.541,-176.611,9.259,148.889
C06712=1138.265,340.132,-79.574,-176.608,9.263,148.889
C06713=1138.261,340.380,-79.608,-176.605,9.268,148.889
C06714=1138.257,340.628,-79.643,-176.603,9.271,148.889
C06715=1138.253,340.875,-79.677,-176.600,9.275,148.890
C06716=1138.249,341.123,-79.711,-176.597,9.279,148.890
C06717=1138.245,341.371,-79.745,-176.595,9.283,148.891
C06718=1138.241,341.618,-79.779,-176.593,9.287,148.891
C06719=1138.237,341.865,-79.813,-176.590,9.291,148.891
C06720=1138.233,342.113,-79.848,-176.588,9.295,148.891
C06721=1138.229,342.360,-79.882,-176.585,9.299,148.892
C06722=1138.225,342.608,-79.915,-176.582,9.303,148.892
C06723=1138.221,342.856,-79.950,-176.579,9.307,148.892
C06724=1138.217,343.103,-79.984,-176.577,9.311,148.893
C06725=1138.213,343.351,-80.019,-176.574,9.315,148.893
C06726=1138.209,343.599,-80.053,-176.572,9.319,148.893
C06727=1138.205,343.847,-80.087,-176.570,9.322,148.894
C06728=1138.201,344.094,-80.122,-176.567,9.326,148.894
C06729=1138.197,344.341,-80.156,-176.564,9.331,148.894
C06730=1138.193,344.589,-80.190,-176.562,9.334,148.895
C06731=1138.189,344.836,-80.224,-176.559,9.338,148.895
C06732=1138.185,345.085,-80.259,-176.556,9.343,148.895
C06733=1138.181,345.332,-80.293,-176.554,9.346,148.896
C06734=1138.177,345.580,-80.328,-176.552,9.350,148.896
C06735=1138.173,345.827,-80.362,-176.549,9.355,148.896
C06736=1138.170,346.075,-80.397,-176.546,9.359,148.897
C06737=1138.165,346.322,-80.431,-176.544,9.362,148.897
C06738=1138.161,346.571,-80.466,-176.541,9.366,148.897
C06739=1138.158,346.817,-80.500,-176.539,9.371,148.898
C06740=1138.154,347.065,-80.535,-176.536,9.374,148.898
C06741=1138.150,347.312,-80.569,-176.534,9.378,148.898
C06742=1138.146,347.560,-80.604,-176.531,9.383,148.899
C06743=1138.141,347.808,-80.638,-176.529,9.386,148.899
C06744=1138.138,348.056,-80.673,-176.527,9.390,148.899
C06745=1138.134,348.302,-80.708,-176.524,9.394,148.900
C06746=1138.130,348.551,-80.743,-176.521,9.399,148.900
C06747=1138.125,348.798,-80.777,-176.519,9.402,148.900
C06748=1138.122,349.046,-80.811,-176.516,9.406,148.901
C06749=1138.118,349.293,-80.847,-176.513,9.411,148.901
C06750=1138.114,349.541,-80.881,-176.511,9.415,148.901
C06751=1138.109,349.788,-80.916,-176.509,9.418,148.902
C06752=1138.106,350.035,-80.951,-176.506,9.423,148.902
C06753=1138.102,350.283,-80.986,-176.503,9.427,148.903
C06754=1138.098,350.531,-81.020,-176.501,9.430,148.903
C06755=1138.094,350.778,-81.056,-176.499,9.435,148.903
C06756=1138.090,351.025,-81.090,-176.496,9.439,148.904
C06757=1138.086,351.274,-81.124,-176.493,9.443,148.904
C06758=1138.083,351.521,-81.160,-176.491,9.447,148.904
C06759=1138.078,351.769,-81.194,-176.488,9.451,148.905
C06760=1138.074,352.016,-81.230,-176.486,9.455,148.905
C06761=1138.071,352.263,-81.264,-176.483,9.459,148.905
C06762=1138.067,352.511,-81.299,-176.481,9.463,148.906
C06763=1138.063,352.759,-81.334,-176.478,9.467,148.906
C06764=1138.059,353.006,-81.369,-176.475,9.471,148.906
C06765=1138.055,353.254,-81.404,-176.473,9.476,148.907
C06766=1138.051,353.501,-81.440,-176.471,9.479,148.907
C06767=1138.046,353.749,-81.474,-176.468,9.483,148.907
C06768=1138.043,353.996,-81.510,-176.466,9.488,148.908
C06769=1138.040,354.244,-81.544,-176.463,9.492,148.908
C06770=1138.035,354.491,-81.579,-176.461,9.495,148.909
C06771=1138.032,354.738,-81.615,-176.458,9.500,148.909
C06772=1138.028,354.986,-81.650,-176.456,9.504,148.909
C06773=1138.023,355.233,-81.685,-176.453,9.508,148.910
C06774=1138.020,355.481,-81.720,-176.451,9.512,148.910
C06775=1138.016,355.729,-81.755,-176.448,9.516,148.911
C06776=1138.012,355.976,-81.791,-176.445,9.520,148.911
C06777=1138.008,356.223,-81.826,-176.443,9.524,148.911
C06778=1138.004,356.471,-81.861,-176.440,9.529,148.912
C06779=1138.000,356.719,-81.896,-176.438,9.532,148.912
C06780=1137.996,356.965,-81.931,-176.435,9.536,148.912
C06781=1137.992,357.213,-81.967,-176.433,9.541,148.913
C06782=1137.988,357.461,-82.002,-176.430,9.545,148.913
C06783=1137.985,357.709,-82.037,-176.427,9.549,148.914
C06784=1137.981,357.956,-82.073,-176.426,9.553,148.914
C06785=1137.977,358.203,-82.108,-176.423,9.557,148.914
C06786=1137.973,358.450,-82.144,-176.420,9.561,148.915
C06787=1137.969,358.698,-82.179,-176.418,9.566,148.915
C06788=1137.965,358.946,-82.214,-176.415,9.570,148.916
C06789=1137.961,359.193,-82.249,-176.413,9.573,148.916
C06790=1137.957,359.441,-82.285,-176.410,9.578,148.916
C06791=1137.953,359.688,-82.321,-176.408,9.582,148.917
C06792=1137.949,359.936,-82.356,-176.405,9.586,148.917
C06793=1137.946,360.183,-82.392,-176.402,9.590,148.917
C06794=1137.942,360.430,-82.427,-176.400,9.595,148.918
C06795=1137.938,360.677,-82.463,-176.397,9.599,148.918
C06796=1137.934,360.925,-82.498,-176.395,9.604,148.919
C06797=1137.931,361.172,-82.534,-176.392,9.607,148.919
C06798=1137.926,361.420,-82.570,-176.390,9.611,148.920
C06799=1137.922,361.668,-82.605,-176.387,9.616,148.920
C06800=1137.919,361.915,-82.641,-176.384,9.620,148.920
C06801=1137.915,362.162,-82.676,-176.382,9.624,148.921
C06802=1137.911,362.410,-82.712,-176.379,9.628,148.921
C06803=1137.907,362.657,-82.749,-176.377,9.633,148.922
C06804=1137.903,362.904,-82.784,-176.374,9.637,148.922
C06805=1137.899,363.152,-82.820,-176.371,9.641,148.922
C06806=1137.896,363.399,-82.855,-176.369,9.646,148.923
C06807=1137.892,363.647,-82.891,-176.366,9.650,148.923
C06808=1137.888,363.895,-82.927,-176.363,9.654,148.923
C06809=1137.884,364.141,-82.963,-176.361,9.659,148.924
C06810=1137.880,364.388,-82.998,-176.358,9.663,148.924
C06811=1137.876,364.673,-83.040,-176.356,9.667,148.925
C06812=1137.872,364.957,-83.081,-176.352,9.672,148.925
C06813=1137.867,365.240,-83.123,-176.349,9.677,148.926
C06814=1137.863,365.524,-83.164,-176.346,9.683,148.926
C06815=1137.859,365.772,-83.199,-176.344,9.687,148.927
C06816=1137.855,366.020,-83.235,-176.341,9.691,148.927
C06817=1137.851,366.267,-83.272,-176.338,9.695,148.927
C06818=1137.848,366.514,-83.307,-176.336,9.700,148.928
C06819=1137.843,366.761,-83.343,-176.333,9.704,148.928
C06820=1137.839,367.008,-83.379,-176.330,9.708,148.929
C06821=1137.835,367.256,-83.415,-176.328,9.713,148.929
C06822=1137.831,367.503,-83.451,-176.325,9.717,148.930
C06823=1137.828,367.750,-83.487,-176.323,9.721,148.930
C06824=1137.824,367.998,-83.523,-176.320,9.726,148.930
C06825=1137.820,368.245,-83.560,-176.317,9.730,148.931
C06826=1137.816,368.493,-83.596,-176.315,9.734,148.931
C06827=1137.812,368.740,-83.632,-176.312,9.739,148.932
C06828=1137.808,368.988,-83.668,-176.309,9.743,148.932
C06829=1137.805,369.234,-83.704,-176.307,9.747,148.932
C06830=1137.800,369.482,-83.741,-176.304,9.751,148.933
C06831=1137.797,369.729,-83.777,-176.301,9.756,148.933
C06832=1137.793,369.977,-83.814,-176.299,9.760,148.934
C06833=1137.790,370.224,-83.850,-176.296,9.764,148.934
C06834=1137.786,370.472,-83.887,-176.294,9.768,148.934
C06835=1137.780,370.851,-83.942,-176.290,9.775,148.935
C06836=1137.762,371.992,-84.112,-176.997,11.154,149.479
C06837=1137.758,372.240,-84.150,-176.994,11.156,149.478
C06838=1137.755,372.487,-84.186,-176.991,11.158,149.478
C06839=1137.751,372.734,-84.223,-176.989,11.160,149.478
C06840=1137.747,372.982,-84.260,-176.985,11.163,149.478
C06841=1137.743,373.229,-84.296,-176.983,11.164,149.478
C06842=1137.740,373.476,-84.333,-176.979,11.167,149.477
C06843=1137.736,373.724,-84.370,-176.977,11.169,149.477
C06844=1137.732,373.971,-84.407,-176.974,11.171,149.477
C06845=1137.728,374.218,-84.444,-176.971,11.173,149.477
C06846=1137.724,374.465,-84.480,-176.968,11.176,149.477
C06847=1137.721,374.713,-84.517,-176.966,11.178,149.477
C06848=1137.717,374.959,-84.555,-176.963,11.180,149.477
C06849=1137.710,375.375,-84.616,-176.958,11.184,149.476
C06850=1137.705,375.790,-84.678,-176.953,11.188,149.476
C06851=1137.698,376.205,-84.740,-176.949,11.191,149.476
C06852=1137.691,376.620,-84.802,-176.944,11.195,149.476
C06853=1137.688,376.867,-84.839,-176.942,11.197,149.475
C06854=1137.684,377.114,-84.876,-176.939,11.200,149.475
C06855=1137.680,377.361,-84.913,-176.936,11.201,149.475
C06856=1137.676,377.608,-84.950,-176.933,11.204,149.475
C06857=1137.673,377.856,-84.987,-176.931,11.206,149.475
C06858=1137.669,378.104,-85.024,-176.928,11.208,149.475
C06859=1137.665,378.350,-85.062,-176.925,11.211,149.475
C06860=1137.661,378.597,-85.099,-176.923,11.212,149.475
C06861=1137.657,378.845,-85.136,-176.920,11.214,149.475
C06862=1137.653,379.092,-85.173,-176.918,11.217,149.475
C06863=1137.650,379.339,-85.210,-176.915,11.219,149.475
C06864=1137.647,379.586,-85.247,-176.912,11.222,149.474
C06865=1137.642,379.834,-85.284,-176.910,11.224,149.474
C06866=1137.639,380.080,-85.321,-176.907,11.226,149.474
C06867=1137.635,380.328,-85.359,-176.905,11.228,149.474
C06868=1137.631,380.575,-85.395,-176.902,11.231,149.474
C06869=1137.627,380.822,-85.433,-176.900,11.232,149.474
C06870=1137.624,381.070,-85.470,-176.897,11.234,149.474
C06871=1137.620,381.316,-85.508,-176.894,11.237,149.474
C06872=1137.616,381.564,-85.545,-176.892,11.239,149.474
C06873=1137.612,381.811,-85.582,-176.890,11.241,149.474
C06874=1137.609,382.058,-85.619,-176.888,11.243,149.474
C06875=1137.605,382.305,-85.656,-176.885,11.246,149.474
C06876=1137.601,382.552,-85.694,-176.882,11.248,149.474
C06877=1137.597,382.800,-85.731,-176.880,11.250,149.474
C06878=1137.593,383.046,-85.769,-176.878,11.252,149.473
C06879=1137.590,383.294,-85.806,-176.875,11.255,149.473
C06880=1137.586,383.541,-85.844,-176.874,11.257,149.474
C06881=1137.582,383.788,-85.880,-176.873,11.257,149.474
C06882=1137.579,384.035,-85.918,-176.872,11.259,149.474
C06883=1137.574,384.283,-85.956,-176.871,11.261,149.474
C06884=1137.571,384.530,-85.994,-176.871,11.262,149.474
C06885=1137.567,384.777,-86.031,-176.869,11.264,149.474
C06886=1137.563,385.024,-86.068,-176.869,11.265,149.474
C06887=1137.559,385.272,-86.105,-176.868,11.267,149.475
C06888=1137.556,385.518,-86.143,-176.868,11.267,149.475
C06889=1137.552,385.766,-86.180,-176.867,11.269,149.475
C06890=1137.548,386.013,-86.218,-176.867,11.270,149.475
C06891=1137.544,386.260,-86.255,-176.866,11.272,149.476
C06892=1137.541,386.507,-86.293,-176.865,11.273,149.476
C06893=1137.537,386.754,-86.329,-176.864,11.275,149.476
C06894=1137.534,387.002,-86.367,-176.864,11.276,149.476
C06895=1137.530,387.248,-86.405,-176.863,11.278,149.476
C06896=1137.526,387.495,-86.442,-176.862,11.280,149.477
C06897=1137.522,387.743,-86.480,-176.863,11.281,149.477
C06898=1137.518,387.990,-86.517,-176.862,11.283,149.477
C06899=1137.515,388.237,-86.555,-176.862,11.284,149.478
C06900=1137.511,388.484,-86.593,-176.861,11.286,149.478
C06901=1137.507,388.697,-86.625,-176.860,11.287,149.478
C06902=1137.505,388.910,-86.657,-176.860,11.288,149.478
C06903=1137.501,389.123,-86.689,-176.860,11.290,149.479
C06904=1137.498,389.336,-86.722,-176.860,11.292,149.479
C06905=1137.495,389.549,-86.754,-176.859,11.293,149.479
C06906=1137.492,389.762,-86.787,-176.859,11.294,149.479
C06907=1137.488,389.975,-86.818,-176.859,11.296,149.480
C06908=1137.485,390.188,-86.851,-176.858,11.297,149.480
C06909=1137.481,390.435,-86.888,-176.859,11.299,149.481
C06910=1137.478,390.682,-86.926,-176.858,11.301,149.481
C06911=1137.474,390.929,-86.963,-176.858,11.302,149.481
C06912=1137.471,391.177,-87.001,-176.857,11.304,149.482
C06913=1137.467,391.423,-87.039,-176.858,11.306,149.482
C06914=1137.463,391.670,-87.075,-176.857,11.308,149.483
C06915=1137.459,391.918,-87.113,-176.857,11.309,149.483
C06916=1137.455,392.165,-87.152,-176.857,11.312,149.484
C06917=1137.451,392.412,-87.189,-176.857,11.313,149.484
C06918=1137.448,392.659,-87.226,-176.856,11.315,149.484
C06919=1137.444,392.906,-87.264,-176.857,11.317,149.485
C06920=1137.440,393.153,-87.301,-176.856,11.319,149.485
C06921=1137.437,393.401,-87.339,-176.857,11.321,149.486
C06922=1137.433,393.647,-87.377,-176.856,11.323,149.486
C06923=1137.429,393.895,-87.414,-176.856,11.325,149.487
C06924=1137.425,394.142,-87.452,-176.856,11.327,149.487
C06925=1137.422,394.389,-87.490,-176.857,11.329,149.488
C06926=1137.418,394.637,-87.527,-176.856,11.331,149.488
C06927=1137.414,394.883,-87.564,-176.857,11.333,149.489
C06928=1137.411,395.130,-87.602,-176.857,11.335,149.490
C06929=1137.406,395.378,-87.640,-176.857,11.337,149.490
C06930=1137.402,395.624,-87.677,-176.857,11.339,149.491
C06931=1137.399,395.872,-87.715,-176.857,11.341,149.491
C06932=1137.395,396.119,-87.752,-176.857,11.343,149.492
C06933=1137.392,396.366,-87.790,-176.858,11.345,149.492
C06934=1137.388,396.613,-87.828,-176.858,11.348,149.493
C06935=1137.384,396.860,-87.866,-176.858,11.350,149.494
C06936=1137.380,397.108,-87.903,-176.859,11.352,149.495
C06937=1137.377,397.355,-87.941,-176.859,11.354,149.495
C06938=1137.373,397.601,-87.979,-176.859,11.357,149.496
C06939=1137.370,397.849,-88.016,-176.859,11.359,149.496
C06940=1137.365,398.096,-88.054,-176.860,11.361,149.497
C06941=1137.361,398.343,-88.092,-176.860,11.364,149.498
C06942=1137.358,398.590,-88.129,-176.861,11.366,149.499
C06943=1137.354,398.837,-88.166,-176.861,11.369,149.499
C06944=1137.351,399.084,-88.204,-176.862,11.371,149.500
C06945=1137.346,399.331,-88.242,-176.862,11.373,149.501
C06946=1137.343,399.579,-88.280,-176.863,11.375,149.501
C06947=1137.339,399.826,-88.317,-176.863,11.378,149.502
C06948=1137.336,400.073,-88.355,-176.864,11.380,149.503
C06949=1137.332,400.320,-88.393,-176.864,11.383,149.504
C06950=1137.328,400.567,-88.431,-176.865,11.385,149.505
C06951=1137.324,400.814,-88.468,-176.865,11.388,149.506
C06952=1137.320,401.061,-88.506,-176.866,11.390,149.506
C06953=1137.317,401.308,-88.544,-176.867,11.393,149.507
C06954=1137.313,401.555,-88.581,-176.868,11.395,149.508
C06955=1137.309,401.803,-88.619,-176.868,11.399,149.509
C06956=1137.305,402.050,-88.657,-176.869,11.401,149.510
C06957=1137.302,402.263,-88.690,-176.870,11.404,149.511
C06958=1137.299,402.475,-88.722,-176.871,11.406,149.511
C06959=1137.296,402.689,-88.754,-176.871,11.407,149.512
C06960=1137.292,402.901,-88.787,-176.871,11.410,149.513
C06961=1137.290,403.114,-88.819,-176.872,11.412,149.514
C06962=1137.286,403.327,-88.851,-176.873,11.415,149.514
C06963=1137.284,403.540,-88.884,-176.874,11.418,149.515
C06964=1137.280,403.752,-88.917,-176.875,11.420,149.516
C06965=1137.277,404.000,-88.954,-176.876,11.423,149.517
C06966=1137.272,404.247,-88.992,-176.877,11.426,149.518
C06967=1137.269,404.494,-89.030,-176.878,11.429,149.519
C06968=1137.265,404.741,-89.068,-176.878,11.432,149.520
C06969=1137.262,404.988,-89.106,-176.880,11.434,149.521
C06970=1137.257,405.235,-89.143,-176.880,11.438,149.522
C06971=1137.254,405.483,-89.181,-176.882,11.440,149.523
C06972=1137.250,405.729,-89.219,-176.883,11.444,149.524
C06973=1137.247,405.977,-89.257,-176.884,11.446,149.525
C06974=1137.243,406.223,-89.294,-176.885,11.450,149.527
C06975=1137.239,406.471,-89.332,-176.886,11.453,149.528
C06976=1137.235,406.718,-89.369,-176.888,11.456,149.529
C06977=1137.232,406.965,-89.407,-176.889,11.459,149.530
C06978=1137.228,407.212,-89.445,-176.890,11.462,149.531
C06979=1137.224,407.459,-89.484,-176.891,11.465,149.532
C06980=1137.220,407.707,-89.520,-176.892,11.469,149.533
C06981=1137.217,407.954,-89.558,-176.894,11.471,149.534
C06982=1137.213,408.200,-89.596,-176.895,11.475,149.536
C06983=1137.209,408.448,-89.634,-176.896,11.479,149.537
C06984=1137.205,408.695,-89.672,-176.898,11.481,149.538
C06985=1137.202,408.942,-89.710,-176.900,11.485,149.539
C06986=1137.198,409.189,-89.747,-176.901,11.489,149.541
C06987=1137.194,409.437,-89.785,-176.902,11.491,149.542
C06988=1137.190,409.683,-89.823,-176.904,11.495,149.543
C06989=1137.187,409.930,-89.861,-176.905,11.499,149.544
C06990=1137.183,410.177,-89.898,-176.907,11.502,149.546
C06991=1137.179,410.425,-89.937,-176.909,11.506,149.547
C06992=1137.175,410.672,-89.974,-176.910,11.509,149.548
C06993=1137.172,410.919,-90.012,-176.912,11.513,149.550
C06994=1137.168,411.166,-90.049,-176.913,11.516,149.551
C06995=1137.164,411.413,-90.088,-176.915,11.520,149.552
C06996=1137.161,411.660,-90.125,-176.917,11.523,149.554
C06997=1137.158,411.907,-90.163,-176.918,11.527,149.555
C06998=1137.153,412.154,-90.200,-176.920,11.532,149.557
C06999=1137.149,412.401,-90.238,-176.922,11.535,149.558
C07000=1137.146,412.648,-90.276,-176.924,11.538,149.559
C07001=1137.142,412.895,-90.314,-176.926,11.543,149.561
C07002=1137.139,413.142,-90.352,-176.927,11.547,149.562
C07003=1137.134,413.389,-90.390,-176.930,11.550,149.564
C07004=1137.131,413.637,-90.427,-176.931,11.554,149.565
C07005=1137.127,413.884,-90.465,-176.933,11.558,149.567
C07006=1137.123,414.131,-90.503,-176.935,11.562,149.568
C07007=1137.120,414.378,-90.541,-176.937,11.566,149.570
C07008=1137.116,414.625,-90.579,-176.939,11.570,149.571
C07009=1137.114,414.873,-90.617,-176.941,11.574,149.573
C07010=1137.112,415.119,-90.653,-176.943,11.578,149.574
C07011=1137.111,415.366,-90.692,-176.946,11.582,149.576
C07012=1137.111,415.613,-90.728,-176.948,11.586,149.578
C07013=1137.110,415.827,-90.761,-176.949,11.590,149.579
C07014=1137.111,416.039,-90.792,-176.952,11.594,149.581
C07015=1137.112,416.252,-90.825,-176.953,11.598,149.582
C07016=1137.113,416.465,-90.856,-176.956,11.601,149.584
C07017=1137.116,416.677,-90.888,-176.957,11.605,149.585
C07018=1137.118,416.891,-90.920,-176.960,11.608,149.586
C07019=1137.120,417.103,-90.952,-176.961,11.612,149.588
C07020=1137.125,417.316,-90.983,-176.963,11.616,149.589
C07021=1136.705,417.316,-91.046,-176.956,11.620,149.589
C07022=1136.701,417.103,-91.014,-176.954,11.617,149.587
C07023=1136.698,416.890,-90.983,-176.952,11.613,149.586
C07024=1136.697,416.677,-90.951,-176.950,11.609,149.584
C07025=1136.694,416.464,-90.919,-176.948,11.605,149.583
C07026=1136.693,416.251,-90.887,-176.946,11.602,149.581
C07027=1136.692,416.039,-90.855,-176.944,11.598,149.580
C07028=1136.691,415.826,-90.823,-176.942,11.595,149.579
C07029=1136.692,415.613,-90.791,-176.941,11.591,149.577
C07030=1136.692,415.367,-90.754,-176.938,11.586,149.575
C07031=1136.693,415.120,-90.717,-176.937,11.582,149.574
C07032=1136.695,414.872,-90.679,-176.934,11.579,149.572
C07033=1136.697,414.625,-90.642,-176.932,11.575,149.571
C07034=1136.700,414.378,-90.604,-176.930,11.570,149.569
C07035=1136.703,414.130,-90.566,-176.928,11.566,149.568
C07036=1136.708,413.884,-90.528,-176.927,11.562,149.566
C07037=1136.711,413.636,-90.490,-176.925,11.558,149.565
C07038=1136.715,413.390,-90.452,-176.923,11.555,149.563
C07039=1136.718,413.142,-90.414,-176.921,11.550,149.562
C07040=1136.723,412.896,-90.376,-176.919,11.547,149.560
C07041=1136.726,412.648,-90.339,-176.917,11.542,149.559
C07042=1136.730,412.401,-90.301,-176.916,11.538,149.557
C07043=1136.734,412.153,-90.263,-176.914,11.535,149.556
C07044=1136.738,411.907,-90.225,-176.912,11.531,149.555
C07045=1136.741,411.660,-90.187,-176.911,11.528,149.553
C07046=1136.745,411.413,-90.150,-176.909,11.523,149.552
C07047=1136.749,411.165,-90.111,-176.907,11.521,149.550
C07048=1136.752,410.919,-90.073,-176.906,11.517,149.549
C07049=1136.756,410.671,-90.036,-176.904,11.513,149.548
C07050=1136.760,410.424,-89.999,-176.903,11.509,149.546
C07051=1136.764,410.177,-89.960,-176.901,11.506,149.545
C07052=1136.767,409.930,-89.923,-176.900,11.502,149.544
C07053=1136.771,409.683,-89.885,-176.898,11.498,149.542
C07054=1136.775,409.436,-89.846,-176.897,11.495,149.541
C07055=1136.779,409.188,-89.809,-176.895,11.492,149.540
C07056=1136.782,408.942,-89.772,-176.894,11.488,149.539
C07057=1136.786,408.694,-89.734,-176.893,11.485,149.537
C07058=1136.790,408.448,-89.695,-176.891,11.482,149.536
C07059=1136.793,408.200,-89.658,-176.890,11.478,149.535
C07060=1136.797,407.954,-89.620,-176.889,11.475,149.534
C07061=1136.800,407.706,-89.582,-176.888,11.471,149.533
C07062=1136.805,407.459,-89.545,-176.886,11.468,149.532
C07063=1136.808,407.212,-89.507,-176.885,11.465,149.530
C07064=1136.812,406.965,-89.469,-176.884,11.461,149.529
C07065=1136.815,406.718,-89.431,-176.882,11.459,149.528
C07066=1136.820,406.471,-89.393,-176.881,11.455,149.527
C07067=1136.823,406.224,-89.355,-176.881,11.452,149.526
C07068=1136.827,405.976,-89.318,-176.879,11.449,149.525
C07069=1136.830,405.729,-89.280,-176.878,11.446,149.524
C07070=1136.835,405.482,-89.242,-176.878,11.443,149.523
C07071=1136.838,405.235,-89.204,-176.876,11.440,149.522
C07072=1136.842,404.988,-89.167,-176.875,11.437,149.521
C07073=1136.845,404.741,-89.129,-176.874,11.435,149.520
C07074=1136.849,404.494,-89.092,-176.873,11.431,149.519
C07075=1136.853,404.246,-89.053,-176.872,11.428,149.518
C07076=1136.857,404.000,-89.016,-176.871,11.426,149.517
C07077=1136.860,403.753,-88.978,-176.870,11.422,149.516
C07078=1136.864,403.540,-88.946,-176.869,11.420,149.515
C07079=1136.867,403.327,-88.913,-176.869,11.417,149.514
C07080=1136.870,403.114,-88.880,-176.868,11.415,149.513
C07081=1136.873,402.901,-88.847,-176.868,11.412,149.512
C07082=1136.877,402.688,-88.815,-176.867,11.410,149.512
C07083=1136.880,402.475,-88.783,-176.866,11.408,149.511
C07084=1136.883,402.263,-88.750,-176.866,11.405,149.510
C07085=1136.887,402.050,-88.718,-176.865,11.404,149.509
C07086=1136.890,401.803,-88.680,-176.864,11.400,149.508
C07087=1136.894,401.556,-88.643,-176.863,11.398,149.508
C07088=1136.897,401.309,-88.605,-176.863,11.395,149.507
C07089=1136.901,401.062,-88.567,-176.862,11.393,149.506
C07090=1136.905,400.814,-88.529,-176.862,11.390,149.505
C07091=1136.909,400.567,-88.492,-176.861,11.388,149.504
C07092=1136.912,400.320,-88.454,-176.860,11.385,149.504
C07093=1136.916,400.074,-88.416,-176.860,11.383,149.503
C07094=1136.919,399.826,-88.379,-176.859,11.380,149.502
C07095=1136.924,399.579,-88.341,-176.859,11.378,149.501
C07096=1136.927,399.332,-88.303,-176.859,11.375,149.500
C07097=1136.931,399.085,-88.265,-176.858,11.373,149.500
C07098=1136.934,398.837,-88.228,-176.858,11.370,149.499
C07099=1136.939,398.590,-88.190,-176.857,11.368,149.498
C07100=1136.942,398.343,-88.152,-176.857,11.365,149.497
C07101=1136.946,398.096,-88.114,-176.856,11.364,149.497
C07102=1136.950,397.849,-88.077,-176.856,11.361,149.496
C07103=1136.953,397.602,-88.040,-176.855,11.359,149.495
C07104=1136.958,397.355,-88.001,-176.855,11.356,149.495
C07105=1136.961,397.108,-87.963,-176.855,11.354,149.494
C07106=1136.965,396.861,-87.927,-176.855,11.352,149.493
C07107=1136.968,396.613,-87.889,-176.855,11.349,149.493
C07108=1136.972,396.367,-87.851,-176.854,11.348,149.492
C07109=1136.975,396.119,-87.814,-176.854,11.345,149.492
C07110=1136.980,395.872,-87.776,-176.854,11.343,149.491
C07111=1136.983,395.625,-87.738,-176.854,11.341,149.490
C07112=1136.987,395.378,-87.700,-176.854,11.339,149.490
C07113=1136.991,395.131,-87.663,-176.854,11.337,149.489
C07114=1136.994,394.884,-87.625,-176.854,11.334,149.489
C07115=1136.999,394.637,-87.587,-176.854,11.333,149.488
C07116=1137.002,394.389,-87.550,-176.854,11.330,149.488
C07117=1137.006,394.142,-87.512,-176.854,11.329,149.487
C07118=1137.009,393.895,-87.474,-176.854,11.326,149.486
C07119=1137.013,393.648,-87.438,-176.854,11.325,149.486
C07120=1137.016,393.401,-87.400,-176.854,11.323,149.486
C07121=1137.021,393.154,-87.361,-176.854,11.321,149.485
C07122=1137.025,392.906,-87.325,-176.854,11.319,149.485
C07123=1137.028,392.659,-87.287,-176.854,11.317,149.484
C07124=1137.032,392.413,-87.249,-176.854,11.315,149.484
C07125=1137.035,392.165,-87.212,-176.855,11.313,149.483
C07126=1137.039,391.918,-87.174,-176.855,11.311,149.483
C07127=1137.042,391.671,-87.136,-176.855,11.309,149.482
C07128=1137.047,391.423,-87.099,-176.855,11.308,149.482
C07129=1137.051,391.177,-87.061,-176.855,11.305,149.481
C07130=1137.054,390.930,-87.023,-176.856,11.304,149.481
C07131=1137.058,390.682,-86.987,-176.856,11.302,149.481
C07132=1137.062,390.435,-86.949,-176.856,11.300,149.480
C07133=1137.065,390.189,-86.911,-176.857,11.299,149.480
C07134=1137.069,389.975,-86.879,-176.857,11.297,149.480
C07135=1137.072,389.763,-86.846,-176.857,11.295,149.479
C07136=1137.075,389.549,-86.814,-176.858,11.294,149.479
C07137=1137.079,389.336,-86.781,-176.857,11.293,149.479
C07138=1137.081,389.123,-86.750,-176.858,11.291,149.478
C07139=1137.085,388.911,-86.717,-176.859,11.290,149.478
C07140=1137.088,388.697,-86.685,-176.859,11.289,149.478
C07141=1137.091,388.485,-86.652,-176.860,11.287,149.478
C07142=1137.095,388.238,-86.615,-176.860,11.286,149.478
C07143=1137.099,387.990,-86.577,-176.860,11.283,149.477
C07144=1137.102,387.744,-86.540,-176.861,11.282,149.477
C07145=1137.106,387.496,-86.503,-176.861,11.280,149.477
C07146=1137.110,387.249,-86.465,-176.862,11.279,149.476
C07147=1137.114,387.002,-86.428,-176.862,11.277,149.476
C07148=1137.117,386.755,-86.390,-176.863,11.276,149.476
C07149=1137.122,386.507,-86.353,-176.864,11.274,149.476
C07150=1137.125,386.260,-86.315,-176.864,11.272,149.475
C07151=1137.129,386.013,-86.277,-176.865,11.272,149.475
C07152=1137.133,385.766,-86.241,-176.866,11.270,149.475
C07153=1137.136,385.519,-86.203,-176.866,11.269,149.475
C07154=1137.140,385.272,-86.166,-176.867,11.267,149.475
C07155=1137.143,385.025,-86.128,-176.868,11.266,149.474
C07156=1137.147,384.777,-86.091,-176.868,11.264,149.474
C07157=1137.151,384.531,-86.053,-176.870,11.262,149.474
C07158=1137.155,384.283,-86.016,-176.870,11.261,149.474
C07159=1137.158,384.036,-85.979,-176.871,11.260,149.474
C07160=1137.162,383.788,-85.941,-176.872,11.259,149.474
C07161=1137.166,383.542,-85.904,-176.873,11.257,149.473
C07162=1137.170,383.295,-85.867,-176.874,11.256,149.473
C07163=1137.173,383.047,-85.829,-176.876,11.253,149.473
C07164=1137.177,382.800,-85.792,-176.879,11.251,149.473
C07165=1137.182,382.553,-85.754,-176.881,11.249,149.473
C07166=1137.185,382.305,-85.717,-176.884,11.247,149.473
C07167=1137.189,382.059,-85.679,-176.886,11.245,149.474
C07168=1137.192,381.811,-85.642,-176.889,11.242,149.474
C07169=1137.196,381.564,-85.604,-176.891,11.240,149.474
C07170=1137.200,381.317,-85.567,-176.893,11.238,149.474
C07171=1137.204,381.069,-85.530,-176.897,11.235,149.474
C07172=1137.208,380.823,-85.493,-176.899,11.233,149.474
C07173=1137.211,380.576,-85.456,-176.901,11.231,149.474
C07174=1137.214,380.328,-85.419,-176.904,11.228,149.474
C07175=1137.218,380.081,-85.382,-176.906,11.226,149.474
C07176=1137.222,379.834,-85.345,-176.909,11.224,149.474
C07177=1137.226,379.587,-85.308,-176.912,11.222,149.474
C07178=1137.230,379.340,-85.270,-176.914,11.220,149.474
C07179=1137.234,379.093,-85.233,-176.916,11.218,149.474
C07180=1137.238,378.845,-85.196,-176.919,11.215,149.474
C07181=1137.241,378.598,-85.158,-176.922,11.213,149.475
C07182=1137.245,378.351,-85.121,-176.924,11.211,149.475
C07183=1137.249,378.104,-85.085,-176.927,11.208,149.475
C07184=1137.253,377.856,-85.047,-176.930,11.207,149.475
C07185=1137.256,377.609,-85.010,-176.932,11.205,149.475
C07186=1137.261,377.362,-84.973,-176.935,11.202,149.475
C07187=1137.264,377.115,-84.937,-176.938,11.200,149.475
C07188=1137.267,376.867,-84.899,-176.941,11.197,149.475
C07189=1137.271,376.620,-84.863,-176.943,11.196,149.476
C07190=1137.275,376.407,-84.831,-176.946,11.194,149.476
C07191=1137.277,376.194,-84.798,-176.948,11.192,149.476
C07192=1137.281,375.981,-84.766,-176.951,11.190,149.476
C07193=1137.285,375.768,-84.735,-176.953,11.188,149.476
C07194=1137.287,375.555,-84.703,-176.955,11.186,149.476
C07195=1137.291,375.342,-84.671,-176.958,11.184,149.476
C07196=1137.294,375.129,-84.640,-176.960,11.182,149.476
C07197=1137.297,374.916,-84.608,-176.962,11.180,149.476
C07198=1137.302,374.669,-84.571,-176.965,11.178,149.477
C07199=1137.306,374.421,-84.534,-176.968,11.176,149.477
C07200=1137.309,374.175,-84.498,-176.971,11.174,149.477
C07201=1137.313,373.927,-84.461,-176.974,11.171,149.477
C07202=1137.317,373.679,-84.424,-176.977,11.170,149.477
C07203=1137.321,373.432,-84.387,-176.979,11.167,149.477
C07204=1137.324,373.185,-84.350,-176.983,11.164,149.478
C07205=1137.328,372.938,-84.314,-176.985,11.163,149.478
C07206=1137.332,372.691,-84.277,-176.988,11.160,149.478
C07207=1137.336,372.443,-84.239,-176.991,11.158,149.478
C07208=1137.339,372.196,-84.203,-176.994,11.156,149.478
C07209=1137.343,371.949,-84.166,-176.997,11.154,149.479
C07210=1137.347,371.702,-84.129,-177.000,11.151,149.479
C07211=1137.351,371.455,-84.093,-177.003,11.149,149.479
C07212=1137.355,371.208,-84.056,-177.006,11.147,149.479
C07213=1137.358,370.960,-84.019,-177.009,11.145,149.479
C07214=1137.362,370.713,-83.983,-177.012,11.143,149.480
C07215=1137.366,370.465,-83.947,-177.015,11.140,149.480
C07216=1137.370,370.218,-83.910,-177.018,11.138,149.480
C07217=1137.373,369.971,-83.874,-177.021,11.136,149.480
C07218=1137.377,369.724,-83.837,-177.024,11.133,149.480
C07219=1137.382,369.477,-83.800,-177.027,11.131,149.480
C07220=1137.385,369.229,-83.764,-177.030,11.129,149.481
C07221=1137.389,368.981,-83.727,-177.033,11.127,149.481
C07222=1137.392,368.734,-83.691,-177.037,11.124,149.481
C07223=1137.396,368.487,-83.654,-177.039,11.123,149.481
C07224=1137.401,368.239,-83.618,-177.043,11.120,149.482
C07225=1137.404,367.993,-83.582,-177.046,11.118,149.482
C07226=1137.408,367.745,-83.545,-177.049,11.115,149.482
C07227=1137.411,367.499,-83.508,-177.052,11.114,149.482
C07228=1137.416,367.251,-83.472,-177.055,11.111,149.482
C07229=1137.419,367.004,-83.436,-177.058,11.109,149.483
C07230=1137.424,366.756,-83.400,-177.062,11.106,149.483
C07231=1137.428,366.509,-83.363,-177.064,11.104,149.483
C07232=1137.431,366.262,-83.327,-177.068,11.102,149.483
C07233=1137.435,366.013,-83.290,-177.071,11.099,149.484
C07234=1137.438,365.767,-83.254,-177.074,11.097,149.484
C07235=1137.443,365.519,-83.218,-177.078,11.095,149.484
C07236=1137.446,365.272,-83.182,-177.081,11.092,149.484
C07237=1137.450,365.025,-83.145,-177.084,11.090,149.484
C07238=1137.454,364.777,-83.109,-177.087,11.088,149.485
C07239=1137.457,364.530,-83.073,-177.091,11.086,149.485
C07240=1137.461,364.282,-83.037,-177.094,11.083,149.485
C07241=1137.465,364.036,-83.001,-177.097,11.081,149.485
C07242=1137.469,363.788,-82.964,-177.100,11.078,149.486
C07243=1137.473,363.541,-82.928,-177.104,11.076,149.486
C07244=1137.476,363.293,-82.893,-177.107,11.073,149.486
C07245=1137.481,363.046,-82.856,-177.111,11.071,149.487
C07246=1137.485,362.775,-82.817,-177.114,11.069,149.487
C07247=1137.489,362.503,-82.777,-177.117,11.066,149.487
C07248=1137.493,362.231,-82.738,-177.122,11.063,149.487
C07249=1137.497,361.960,-82.698,-177.125,11.061,149.488
C07250=1137.501,361.712,-82.662,-177.129,11.059,149.488
C07251=1137.505,361.465,-82.626,-177.132,11.056,149.488
C07252=1137.508,361.218,-82.590,-177.135,11.054,149.488
C07253=1137.513,360.970,-82.554,-177.139,11.051,149.489
C07254=1137.530,359.814,-82.386,-176.409,9.595,148.920
C07255=1137.537,359.430,-82.330,-176.412,9.589,148.920
C07256=1137.541,359.181,-82.296,-176.415,9.585,148.919
C07257=1137.544,358.934,-82.260,-176.417,9.580,148.919
C07258=1137.548,358.686,-82.225,-176.420,9.576,148.919
C07259=1137.552,358.439,-82.189,-176.423,9.572,148.918
C07260=1137.556,358.192,-82.154,-176.425,9.568,148.918
C07261=1137.559,357.945,-82.118,-176.427,9.564,148.917
C07262=1137.564,357.697,-82.082,-176.430,9.560,148.917
C07263=1137.568,357.449,-82.047,-176.433,9.556,148.917
C07264=1137.572,357.202,-82.012,-176.435,9.551,148.916
C07265=1137.576,356.954,-81.977,-176.437,9.548,148.916
C07266=1137.579,356.707,-81.941,-176.440,9.544,148.916
C07267=1137.583,356.459,-81.905,-176.443,9.539,148.915
C07268=1137.588,356.212,-81.871,-176.445,9.535,148.915
C07269=1137.591,355.964,-81.835,-176.448,9.530,148.914
C07270=1137.595,355.717,-81.800,-176.450,9.527,148.914
C07271=1137.599,355.469,-81.765,-176.452,9.523,148.914
C07272=1137.603,355.222,-81.731,-176.455,9.518,148.913
C07273=1137.606,354.975,-81.695,-176.458,9.514,148.913
C07274=1137.610,354.727,-81.660,-176.460,9.510,148.912
C07275=1137.614,354.480,-81.625,-176.462,9.506,148.912
C07276=1137.618,354.232,-81.589,-176.465,9.502,148.912
C07277=1137.622,353.984,-81.555,-176.468,9.498,148.911
C07278=1137.626,353.738,-81.519,-176.470,9.494,148.911
C07279=1137.630,353.489,-81.485,-176.473,9.490,148.911
C07280=1137.634,353.242,-81.449,-176.475,9.486,148.910
C07281=1137.638,352.994,-81.415,-176.478,9.482,148.910
C07282=1137.642,352.747,-81.379,-176.481,9.478,148.909
C07283=1137.645,352.499,-81.345,-176.483,9.474,148.909
C07284=1137.650,352.252,-81.310,-176.485,9.470,148.909
C07285=1137.654,352.004,-81.275,-176.488,9.465,148.908
C07286=1137.657,351.757,-81.239,-176.491,9.461,148.908
C07287=1137.662,351.509,-81.205,-176.493,9.458,148.908
C07288=1137.666,351.262,-81.169,-176.495,9.453,148.907
C07289=1137.669,351.015,-81.135,-176.498,9.449,148.907
C07290=1137.673,350.767,-81.100,-176.501,9.445,148.907
C07291=1137.677,350.519,-81.065,-176.503,9.441,148.906
C07292=1137.682,350.272,-81.030,-176.506,9.437,148.906
C07293=1137.685,350.024,-80.995,-176.508,9.433,148.905
C07294=1137.689,349.777,-80.961,-176.511,9.429,148.905
C07295=1137.693,349.529,-80.926,-176.513,9.425,148.905
C07296=1137.697,349.282,-80.891,-176.516,9.421,148.904
C07297=1137.701,349.034,-80.856,-176.519,9.417,148.904
C07298=1137.704,348.786,-80.822,-176.521,9.413,148.904
C07299=1137.709,348.539,-80.787,-176.523,9.409,148.903
C07300=1137.713,348.291,-80.752,-176.526,9.405,148.903
C07301=1137.717,348.044,-80.718,-176.528,9.400,148.903
C07302=1137.721,347.796,-80.683,-176.531,9.397,148.902
C07303=1137.725,347.549,-80.649,-176.533,9.393,148.902
C07304=1137.728,347.301,-80.614,-176.536,9.389,148.902
C07305=1137.733,347.054,-80.579,-176.539,9.384,148.901
C07306=1137.737,346.806,-80.545,-176.541,9.381,148.901
C07307=1137.740,346.559,-80.511,-176.544,9.377,148.901
C07308=1137.744,346.311,-80.476,-176.547,9.373,148.900
C07309=1137.749,346.063,-80.441,-176.548,9.369,148.900
C07310=1137.752,345.815,-80.407,-176.551,9.365,148.900
C07311=1137.757,345.568,-80.373,-176.554,9.361,148.899
C07312=1137.760,345.321,-80.337,-176.557,9.357,148.899
